// TwinCAT 3 PLC project Plc_Prog
// ProgramVersion: 3.1.4024.0
// libraries:
//   CPNTeck - OSCAT BASIC, * (CPNTeck - Automação Industrial)
//   Tc2_EtherCAT, * (Beckhoff Automation GmbH)
//   Tc2_ModbusSrv, * (Beckhoff Automation GmbH)
//   Tc2_Standard, * (Beckhoff Automation GmbH)
//   Tc2_SUPS, * (Beckhoff Automation GmbH)
//   Tc2_System, * (Beckhoff Automation GmbH)
//   Tc2_Utilities, * (Beckhoff Automation GmbH)
//   Tc3_Module, * (Beckhoff Automation GmbH)
// project tree:
//   Function Blocks/DELTA - MS300/ C2000_ANALOG_INPUTS.TcDUT, C2000_ANALOG_OUTPUTS.TcDUT, C2000_CONTROLWORD.TcDUT, C2000_DEV_CONFIG.TcDUT (not stored), C2000_DIGITAL_INPUTS.TcDUT (not stored), C2000_DIGITAL_OUTPUTS.TcDUT, C2000_DRVTOPLC_PDOS.TcDUT, C2000_PDOS.TcDUT (not stored), C2000_PLCTODRV_PDOS.TcDUT, C2000_STATUSWORD.TcDUT, E_C2000_ModeOfOperation.TcDUT (not stored), FB_DELTA_C2000_ETC.TcPOU
//   Function Blocks/IOs/Beckhoff/Common/ FB_SavePersistentData.TcPOU
//   Function Blocks/IOs/Beckhoff/EL1809 - Digital Inputs/DataTypes/ EL1809_DEV_CONFIG.TcDUT (not stored), EL1809_HWTOPLC_PDOS.TcDUT, EL1809_PDOS.TcDUT (not stored)
//   Function Blocks/IOs/Beckhoff/EL1809 - Digital Inputs/ FB_EL1809.TcPOU (not stored)
//   Function Blocks/IOs/Beckhoff/EL3052 - Ai 2 x 4-20MA - 12bit/DataTypes/ EL3052_DEV_CONFIG.TcDUT, EL3052_DEV_STATUS.TcDUT, EL3052_HWTOPLC_PDOS.TcDUT, EL3052_CHANNEL.TcDUT (not stored), EL3052_PDOS.TcDUT (not stored)
//   Function Blocks/IOs/Beckhoff/EL3052 - Ai 2 x 4-20MA - 12bit/ FB_EL3052.TcPOU
//   Function Blocks/IOs/Beckhoff/EL2809 - Digital Outputs/DataTypes/ EL2809_DEV_CONFIG.TcDUT, EL2809_PDOS.TcDUT (not stored), EL2809_PLCTOHW_PDOS.TcDUT
//   Function Blocks/IOs/Beckhoff/EL2809 - Digital Outputs/ FB_EL2809.TcPOU (not stored)
//   Function Blocks/IOs/Beckhoff/EL3152 - Ai 2 x 4-20MA - 16bit/DataTypes/ EL3152_CHANNEL.TcDUT, EL3152_DEV_CONFIG.TcDUT, EL3152_DEV_STATUS.TcDUT, EL3152_HWTOPLC_PDOS.TcDUT (not stored), EL3152_PDOS.TcDUT
//   Function Blocks/IOs/Beckhoff/EL3152 - Ai 2 x 4-20MA - 16bit/ FB_EL3152.TcPOU (not stored)
//   Function Blocks/IOs/Beckhoff/EL3154 - Ai 4 x 4-20MA - 16bit/DataTypes/ EL3154_CHANNEL.TcDUT (not stored), EL3154_DEV_CONFIG.TcDUT, EL3154_DEV_STATUS.TcDUT, EL3154_HWTOPLC_PDOS.TcDUT (not stored), EL3154_PDOS.TcDUT
//   Function Blocks/IOs/Beckhoff/EL3154 - Ai 4 x 4-20MA - 16bit/ FB_EL3154.TcPOU
//   Function Blocks/IOs/Beckhoff/EL3204 - Ai 4 x PT100 %28RTD%29/DataTypes/ EL3204_DEV_CONFIG.TcDUT (not stored), EL3204_CHANNEL.TcDUT (not stored), EL3204_DEV_STATUS.TcDUT (not stored), EL3204_HWTOPLC_PDOS.TcDUT (not stored), EL3204_PDOS.TcDUT (not stored)
//   Function Blocks/IOs/Beckhoff/EL3204 - Ai 4 x PT100 %28RTD%29/ FB_EL3204.TcPOU (not stored)
//   Function Blocks/IOs/Beckhoff/EL4004 - AQ 4 x 0-10V/DataTypes/ EL4004_DEV_CONFIG.TcDUT, EL4004_HWTOPLC_PDOS.TcDUT, EL4004_PDOS.TcDUT
//   Function Blocks/IOs/Beckhoff/EL4004 - AQ 4 x 0-10V/ FB_EL4004.TcPOU
//   Function Blocks/IOs/Beckhoff/EL4024 - AQ 4 x 4-20MA/DataTypes/ EL4024_DEV_CONFIG.TcDUT, EL4024_HWTOPLC_PDOS.TcDUT, EL4024_PDOS.TcDUT
//   Function Blocks/IOs/Beckhoff/EL4024 - AQ 4 x 4-20MA/ FB_EL4024.TcPOU
//   Function Blocks/IOs/Beckhoff/EL6910 - TwinSAFE PLC/ EL6910_ESTOP.TcDUT, EL6910_ESTOP_DIGNOSTICS.TcDUT, EL6910_ESTOP_STATUS.TcDUT (not stored), EL6910_HWTOPLC_PDOS.TcDUT, EL6910_PDOS.TcDUT (not stored), EL6910_PLCTOHW_PDOS.TcDUT (not stored), FB_EL6910.TcPOU
//   Function Blocks/PaperMachine/Auxiliary/ FB_FormingBoardDriveControl.TcPOU (not stored), FB_ConsistencyControllerModbusTcp.TcPOU, FB_FormingBoardRollUpDown.TcPOU (not stored), FB_FormingBoardWireStretchControl.TcPOU, FB_Gen_SRamp.TcPOU, FB_HeadboxLipsPWMControl.TcPOU, FB_JumboWeightCapture.TcPOU, FB_LevelControl.TcPOU (not stored), FB_LevelControl_V2.TcPOU, FB_MixPumpControl.TcPOU (not stored), FB_MixPumpControl_V1.TcPOU (not stored), FB_PaperMachine.TcPOU (not stored), FB_PressureControl.TcPOU, FB_PressureControl_V1.TcPOU (not stored), FB_StockPumpFlowControl.TcPOU, FB_VfdProcessControler.TcPOU (not stored), FB_ValveProcessControler.TcPOU, FB_SimpleMotorStart.TcPOU (not stored), FB_SimpleMotorStart_V2.TcPOU (not stored), FB_SimpleMotorStart_V3.TcPOU, FB_SoftstarterSimple.TcPOU, FB_SoftstarterWithBypass.TcPOU (not stored), FB_SoftstarterWithBypass_V1.TcPOU (not stored), FB_SpeedDroopControl.TcPOU (not stored), FB_SpeedDroopControl_1.TcPOU (not stored), FB_WirePitControl.TcPOU, FB_WirePitControl_1.TcPOU
//   Function Blocks/PaperMachine/DataTypes/ PaperMachine_TypeHmiConfig.TcDUT, PaperMachine_TypeHmiCommands.TcDUT, PaperMachine_TypeHmiStatus.TcDUT, PaperMachine_TypeHmiAlarms.TcDUT, ST_ConsistencyControllerConfig.TcDUT, ST_ConsistencyControllerInputs.TcDUT
//   Function Blocks/PaperMachine/DriveControl/ FB_DryingSectionDriveControl_V1.TcPOU, FB_DryingSectionDriveControl_V2.TcPOU, FB_DryingSectionDriveControl_V3.TcPOU (not stored), FB_FormingBoardControl_V3.TcPOU, FB_PressSectionDriveControl_V2_bak.TcPOU (not stored), FB_WinderDriveControl_V1.TcPOU (not stored), FB_DryingSectionLubrificationControl_V1.TcPOU (not stored), FB_DryingSectionPressureControl.TcPOU, FB_FormingBoardControl_V1.TcPOU (not stored), FB_PressSectionDriveControl_V1.TcPOU, FB_PressSectionDriveControl_V2.TcPOU
//   Function Blocks/PaperMachine/ FB_AlarmControl.TcPOU (not stored), FB_GroupDisplayFilters_V1.TcPOU (not stored), FB_GroupDriveControl_V1.TcPOU, FB_GroupSpeedControl_V1.TcPOU (not stored), FB_FormingBoardSpeedControl.TcPOU, FB_DryingSecSpeedControl.TcPOU (not stored), FB_WinderSpeedControl.TcPOU (not stored), FB_GroupTorqueTrimControl_V1.TcPOU (not stored), FB_GroupTorqueTrimControl_V2.TcPOU
//   Function Blocks/Rewinder/DataTypes/ RewinderConfig_TypeStruct.TcDUT, Rewinder_TypePressRoll.TcDUT (not stored), Rewinder_TypeBrakeControl.TcDUT (not stored)
//   Function Blocks/Rewinder/ FB_RewinderControl_V1.TcPOU
//   GVLs/ GVL_Hw.TcGVL
//   / PlcTask.TcTTO, RecipeManager.TcRMO (not stored)
//   POUs/Implicit Checks/ CheckBounds.TcPOU, CheckDivDInt.TcPOU (not stored), CheckDivLInt.TcPOU (not stored), CheckDivLReal.TcPOU, CheckDivReal.TcPOU, CheckLRangeSigned.TcPOU, CheckLRangeUnsigned.TcPOU, CheckPointer.TcPOU, CheckRangeSigned.TcPOU, CheckRangeUnsigned.TcPOU (not stored)
//   POUs/ MAIN.TcPOU
// real-time tasks:
//   TASK PlcTask: cycle T#5ms, priority 20, ADS port 350
// I/O:
//   DEVICE ETH, AmsNetId 192.168.100.1.3.1
//     +P5=050-BC1 - PLC Cabinet [EK1100 EtherCAT Coupler (2A E-Bus)]
//       +P5=050-DI1 (EL1809) [EL1809 16Ch. Dig. Input 24V, 3ms]
//       +P5=050-DI2 (EL1809) [EL1809 16Ch. Dig. Input 24V, 3ms]
//       +P5=050-DI3 (EL1809) [EL1809 16Ch. Dig. Input 24V, 3ms]
//       +P5=050-DO1 (EL2809) [EL2809 16Ch. Dig. Output 24V, 0.5A]
//       +P5=050-DO2 (EL2809) [EL2809 16Ch. Dig. Output 24V, 0.5A]
//       +P5=050-DO3 (EL2809) [EL2809 16Ch. Dig. Output 24V, 0.5A]
//       +P5=050-SP1 (EL6910) [EL6910, TwinSAFE PLC]
//       +P5=050-SI1 (EL1918) [EL1918, 8Ch. Safety Input 24V, TwinSAFE]
//         modules: Module 1 (FSOE), Module 2 (FSLOGIC)
//       +P5=050-SO1 (EL2904) [EL2904, 4 Ch. Safety Output 24V, 0.5A, TwinSAFE]
//         modules: Module 1 (FSOES), Module 2 (DO)
//       +P5=050-SO2 (EL2904) [EL2904, 4 Ch. Safety Output 24V, 0.5A, TwinSAFE]
//         modules: Module 1 (FSOES), Module 2 (DO)
//       +P5=050-BC2 [EL6601 1 Port Switch (Ethernet, CoE)]
//       +P5=050-BC3 [EL6601 1 Port Switch (Ethernet, CoE)]
//       +P5=050-BE1 [EL9011 End Terminal]
//     +P5=050-BC2 - PLC Cabinet [EK1100 EtherCAT Coupler (2A E-Bus)]
//       +P5=050-AI (EL3052) [EL3052 2Ch. Ana. Input 4-20mA]
//       +P5=050-AI2 (EL3152) [EL3152 2Ch. Ana Input 4-20mA]
//       +P5=050-AI3 (EL3052) [EL3052 2Ch. Ana. Input 4-20mA]
//       +P5=050-AI4 (EL3052) [EL3052 2Ch. Ana. Input 4-20mA]
//       +P5=050-BE2 [EL9011 End Terminal]
//     +P4=300-UG1 - Mix Pump [Delta CH2000 EtherCAT(CoE)]
//     +P3=300-UG1 - WirePit Pump [Delta CH2000 EtherCAT(CoE)]
//     +P3=100-UG1 - SuctionRoll [Delta CH2000 EtherCAT(CoE)]
//     +P3=100-UG1 - CouchPit [Delta CH2000 EtherCAT(CoE)]
//     +P3=100-UG2 - Stock pump [Delta CH2000 EtherCAT(CoE)]
//     +P2=100-UG1 - Drive Roll [Delta CH2000 EtherCAT(CoE)]
//     +P9=050-BC1 - Vaccum PLC Cabinet [EK1100 EtherCAT Coupler (2A E-Bus)]
//       +P9=050-DI1 (EL1809) [EL1809 16Ch. Dig. Input 24V, 3ms]
//       +P9=050-DI2 (EL1809) [EL1809 16Ch. Dig. Input 24V, 3ms]
//       +P9=050-DI3 (EL1809) [EL1809 16Ch. Dig. Input 24V, 3ms]
//       +P9=050-DO1 (EL2809) [EL2809 16Ch. Dig. Output 24V, 0.5A]
//       +P9=050-DO2 (EL2809) [EL2809 16Ch. Dig. Output 24V, 0.5A]
//       +P9=050-DO3 (EL2809) [EL2809 16Ch. Dig. Output 24V, 0.5A]
//       +P9=050-AI1 (EL3054) [EL3054 4Ch. Ana. Input 4-20mA]
//       Term 101 (EL3052) [EL3052 2Ch. Ana. Input 4-20mA]
//       Term 102 (EL4004) [EL4004 4Ch. Ana. Output 0-10V, 12bit]
//       Term 151 (EL9011) [EL9011 End Terminal]
//       +P9=050-BE1 [EL9011 End Terminal]
//     +P10=050-BC1 - Press / Dryer PLC Cabinet [EK1100 EtherCAT Coupler (2A E-Bus)]
//       +P10=050-DI1 (EL1809) [EL1809 16Ch. Dig. Input 24V, 3ms]
//       +P10=050-DI2 (EL1809) [EL1809 16Ch. Dig. Input 24V, 3ms]
//       +P10=050-DI3 (EL1809) [EL1809 16Ch. Dig. Input 24V, 3ms]
//       +P10=050-DI4 (EL1809) [EL1809 16Ch. Dig. Input 24V, 3ms]
//       +P10=050-DI5 (EL1809) [EL1809 16Ch. Dig. Input 24V, 3ms]
//       +P10=050-DI6 (EL1809) [EL1809 16Ch. Dig. Input 24V, 3ms]
//       +P10=050-DI7 (EL1809) [EL1809 16Ch. Dig. Input 24V, 3ms]
//       +P10=050-DI8 (EL1809) [EL1809 16Ch. Dig. Input 24V, 3ms]
//       +P10=050-DO1 (EL2809) [EL2809 16Ch. Dig. Output 24V, 0.5A]
//       +P10=050-DO2 (EL2809) [EL2809 16Ch. Dig. Output 24V, 0.5A]
//       +P10=050-DO3 (EL2809) [EL2809 16Ch. Dig. Output 24V, 0.5A]
//       +P10=050-DO4 (EL2809) [EL2809 16Ch. Dig. Output 24V, 0.5A]
//       +P10=050-SI1 (EL1918) [EL1918, 8Ch. Safety Input 24V, TwinSAFE]
//         modules: Module 1 (FSOE), Module 2 (FSLOGIC)
//       +P10=050-SO1 (EL2904) [EL2904, 4 Ch. Safety Output 24V, 0.5A, TwinSAFE]
//         modules: Module 1 (FSOES), Module 2 (DO)
//       +P10=050-BE1 [EL9011 End Terminal]
//     +P10=050-BC2 - Press / Dryer PLC Cabinet [EK1100 EtherCAT Coupler (2A E-Bus)]
//       +P10=050-AI1 (EL3054) [EL3054 4Ch. Ana. Input 4-20mA]
//       +P10=050-AI2 (EL3204) [EL3204 4Ch. Ana. Input PT100 (RTD)]
//       +P10=050-AO1(EL4024) [EL4024 4Ch. Ana. Output 4-20mA, 12bit]
//       +P10=050-BE2 [EL9011 End Terminal]
//     +P11=400-UG1 - Second Press [Delta C2000Plus EtherCAT(CoE)]
//     +P12=400-UG1 - First Press [Delta C2000Plus EtherCAT(CoE)]
//     +P13=500-UG1 - Dryer Section GR1 - Upper GR1 Slave [Delta C2000Plus EtherCAT(CoE)]
//     +P12=500-UG2 - Dryer Section GR1 - Lower GR1 Master [Delta C2000Plus EtherCAT(CoE)]
//     +P12=500-UG3 - Dryer Section GR1 - Upper Master [Delta CH2000 EtherCAT(CoE)]
//     +P12=501-UG1 - Dryer Section  GR2 - Lower Slave [Delta C2000Plus EtherCAT(CoE)]
//     +P12=501-UG2 - Dryer Section GR2 - Upper Slave [Delta CH2000 EtherCAT(CoE)]
//     +P12=501-UG3 - Dryer Section GR2 - Lower Master [Delta C2000Plus EtherCAT(CoE)]
//     +P13=501-UG1 - Dryer Section GR2 - Upper Master [Delta CH2000 EtherCAT(CoE)]
//     +P13=502-UG2 - Dryer Section GR3 - Lower Slave [Delta C2000Plus EtherCAT(CoE)]
//     +P13=502-UG2 - Dryer Section GR3 - Upper Slave [Delta C2000Plus EtherCAT(CoE)]
//     +P13=502-UG3 - Dryer Section GR3 - Lower Master [Delta C2000Plus EtherCAT(CoE)]
//     +P13=502-UG4 - Dryer Section GR3 - Upper Master [Delta C2000Plus EtherCAT(CoE)]
//     +P14=600-UG1 - Winder [Delta C2000Plus EtherCAT(CoE)]
//     +CP2=050-BC1 - Winder command panel [EK1100 EtherCAT Coupler (2A E-Bus)]
//       +CP2=050-SI1 (EL1918) [EL1918, 8Ch. Safety Input 24V, TwinSAFE]
//         modules: Module 1 (FSOE), Module 2 (FSLOGIC)
//       +CP2=050-DI1 (EL1809) [EL1809 16Ch. Dig. Input 24V, 3ms]
//       +CP2=050-DO1 (EL2809 [EL2809 16Ch. Dig. Output 24V, 0.5A]
//       +CP2=050-AO1 (EL4024) [EL4024 4Ch. Ana. Output 4-20mA, 12bit]
//       +CP2=050-BE1 (EL4024) [EL9011 End Terminal]
// variable links:
//   ETH <-> ETH/+CP2=050-BC1 - Winder command panel/+CP2=050-SI1 (EL1918)
//     +P5=050-BC1 - PLC Cabinet/+P5=050-SP1 (EL6910)/ConnectionInputs/TwinSafeGroup1.+CP2=050-SI1 (EL1918) - Module 1 (FSOE)_9 TxPDO <-> Module 1 (FSOE)/FSoE Outputs/FSOE
//     +P5=050-BC1 - PLC Cabinet/+P5=050-SP1 (EL6910)/ConnectionOutputs/TwinSafeGroup1.+CP2=050-SI1 (EL1918) - Module 1 (FSOE)_9 RxPDO <-> Module 1 (FSOE)/FSoE Inputs/FSOE
//   ETH <-> ETH/+P10=050-BC1 - Press / Dryer PLC Cabinet/+P10=050-SI1 (EL1918)
//     +P5=050-BC1 - PLC Cabinet/+P5=050-SP1 (EL6910)/ConnectionInputs/TwinSafeGroup1.+P10=050-SI1 (EL1918) - Module 1 (FSOE)_7 TxPDO <-> Module 1 (FSOE)/FSoE Outputs/FSOE
//   ETH <-> ETH/+P10=050-BC1 - Press / Dryer PLC Cabinet/+P10=050-SO1 (EL2904)
//     +P5=050-BC1 - PLC Cabinet/+P5=050-SP1 (EL6910)/ConnectionInputs/TwinSafeGroup1.+P10=050-SO1 (EL2904) - Module 1 (FSOES)_8 TxPDO <-> Module 1 (FSOES)/RxPDO/FSOE
//     +P5=050-BC1 - PLC Cabinet/+P5=050-SP1 (EL6910)/ConnectionOutputs/TwinSafeGroup1.+P10=050-SO1 (EL2904) - Module 1 (FSOES)_8 RxPDO <-> Module 1 (FSOES)/TxPDO/FSOE
//   ETH <-> ETH/+P5=050-BC1 - PLC Cabinet/+P5=050-SI1 (EL1918)
//     +P5=050-BC1 - PLC Cabinet/+P5=050-SP1 (EL6910)/ConnectionInputs/TwinSafeGroup1.Term 9 (EL1918) - Module 1 (FSOE)_3 TxPDO <-> Module 1 (FSOE)/FSoE Outputs/FSOE
//   ETH <-> ETH/+P5=050-BC1 - PLC Cabinet/+P5=050-SP1 (EL6910)
//     +P10=050-BC1 - Press / Dryer PLC Cabinet/+P10=050-SI1 (EL1918)/Module 1 (FSOE)/FSoE Inputs/FSOE <-> ConnectionOutputs/TwinSafeGroup1.+P10=050-SI1 (EL1918) - Module 1 (FSOE)_7 RxPDO
//     +P5=050-BC1 - PLC Cabinet/+P5=050-SI1 (EL1918)/Module 1 (FSOE)/FSoE Inputs/FSOE <-> ConnectionOutputs/TwinSafeGroup1.Term 9 (EL1918) - Module 1 (FSOE)_3 RxPDO
//     +P5=050-BC1 - PLC Cabinet/+P5=050-SO1 (EL2904)/Module 1 (FSOES)/RxPDO/FSOE <-> ConnectionInputs/TwinSafeGroup1.Term 10 (EL2904) - Module 1 (FSOES)_4 TxPDO
//     +P5=050-BC1 - PLC Cabinet/+P5=050-SO2 (EL2904)/Module 1 (FSOES)/RxPDO/FSOE <-> ConnectionInputs/TwinSafeGroup1.Term 11 (EL2904) - Module 1 (FSOES)_5 TxPDO
//     +P5=050-BC1 - PLC Cabinet/+P5=050-SO1 (EL2904)/Module 1 (FSOES)/TxPDO/FSOE <-> ConnectionOutputs/TwinSafeGroup1.Term 10 (EL2904) - Module 1 (FSOES)_4 RxPDO
//     +P5=050-BC1 - PLC Cabinet/+P5=050-SO2 (EL2904)/Module 1 (FSOES)/TxPDO/FSOE <-> ConnectionOutputs/TwinSafeGroup1.Term 11 (EL2904) - Module 1 (FSOES)_5 RxPDO
//   Plc_Prog/Plc_Prog Instance <-> ETH/+CP2=050-BC1 - Winder command panel/+CP2=050-AO1 (EL4024)
//     PlcTask Outputs/.CP1_050_AO1.PDOS.HwToPLC.Channel1 <-> AO Outputs Channel 1/Analog output
//     PlcTask Outputs/.CP1_050_AO1.PDOS.HwToPLC.Channel2 <-> AO Outputs Channel 2/Analog output
//     PlcTask Outputs/.CP1_050_AO1.PDOS.HwToPLC.Channel3 <-> AO Outputs Channel 3/Analog output
//     PlcTask Outputs/.CP1_050_AO1.PDOS.HwToPLC.Channel4 <-> AO Outputs Channel 4/Analog output
//   Plc_Prog/Plc_Prog Instance <-> ETH/+CP2=050-BC1 - Winder command panel/+CP2=050-DI1 (EL1809)
//     PlcTask Inputs/.CP1_050_DI1.PDOS.digitalInput_01 <-> Channel 1/Input
//     PlcTask Inputs/.CP1_050_DI1.PDOS.digitalInput_02 <-> Channel 2/Input
//     PlcTask Inputs/.CP1_050_DI1.PDOS.digitalInput_03 <-> Channel 3/Input
//     PlcTask Inputs/.CP1_050_DI1.PDOS.digitalInput_04 <-> Channel 4/Input
//     PlcTask Inputs/.CP1_050_DI1.PDOS.digitalInput_05 <-> Channel 5/Input
//     PlcTask Inputs/.CP1_050_DI1.PDOS.digitalInput_06 <-> Channel 6/Input
//     PlcTask Inputs/.CP1_050_DI1.PDOS.digitalInput_07 <-> Channel 7/Input
//     PlcTask Inputs/.CP1_050_DI1.PDOS.digitalInput_08 <-> Channel 8/Input
//     PlcTask Inputs/.CP1_050_DI1.PDOS.digitalInput_09 <-> Channel 9/Input
//     PlcTask Inputs/.CP1_050_DI1.PDOS.digitalInput_10 <-> Channel 10/Input
//     PlcTask Inputs/.CP1_050_DI1.PDOS.digitalInput_11 <-> Channel 11/Input
//     PlcTask Inputs/.CP1_050_DI1.PDOS.digitalInput_12 <-> Channel 12/Input
//     PlcTask Inputs/.CP1_050_DI1.PDOS.digitalInput_13 <-> Channel 13/Input
//     PlcTask Inputs/.CP1_050_DI1.PDOS.digitalInput_14 <-> Channel 14/Input
//     PlcTask Inputs/.CP1_050_DI1.PDOS.digitalInput_15 <-> Channel 15/Input
//     PlcTask Inputs/.CP1_050_DI1.PDOS.digitalInput_16 <-> Channel 16/Input
//   Plc_Prog/Plc_Prog Instance <-> ETH/+CP2=050-BC1 - Winder command panel/+CP2=050-DO1 (EL2809
//     PlcTask Outputs/.CP1_050_DO1.PDOS.PlcToHw.digitalOutput_01 <-> Channel 1/Output
//     PlcTask Outputs/.CP1_050_DO1.PDOS.PlcToHw.digitalOutput_02 <-> Channel 2/Output
//     PlcTask Outputs/.CP1_050_DO1.PDOS.PlcToHw.digitalOutput_03 <-> Channel 3/Output
//     PlcTask Outputs/.CP1_050_DO1.PDOS.PlcToHw.digitalOutput_04 <-> Channel 4/Output
//     PlcTask Outputs/.CP1_050_DO1.PDOS.PlcToHw.digitalOutput_05 <-> Channel 5/Output
//     PlcTask Outputs/.CP1_050_DO1.PDOS.PlcToHw.digitalOutput_06 <-> Channel 6/Output
//     PlcTask Outputs/.CP1_050_DO1.PDOS.PlcToHw.digitalOutput_07 <-> Channel 7/Output
//     PlcTask Outputs/.CP1_050_DO1.PDOS.PlcToHw.digitalOutput_08 <-> Channel 8/Output
//     PlcTask Outputs/.CP1_050_DO1.PDOS.PlcToHw.digitalOutput_09 <-> Channel 9/Output
//     PlcTask Outputs/.CP1_050_DO1.PDOS.PlcToHw.digitalOutput_10 <-> Channel 10/Output
//     PlcTask Outputs/.CP1_050_DO1.PDOS.PlcToHw.digitalOutput_11 <-> Channel 11/Output
//     PlcTask Outputs/.CP1_050_DO1.PDOS.PlcToHw.digitalOutput_12 <-> Channel 12/Output
//     PlcTask Outputs/.CP1_050_DO1.PDOS.PlcToHw.digitalOutput_13 <-> Channel 13/Output
//     PlcTask Outputs/.CP1_050_DO1.PDOS.PlcToHw.digitalOutput_14 <-> Channel 14/Output
//     PlcTask Outputs/.CP1_050_DO1.PDOS.PlcToHw.digitalOutput_15 <-> Channel 15/Output
//     PlcTask Outputs/.CP1_050_DO1.PDOS.PlcToHw.digitalOutput_16 <-> Channel 16/Output
//   Plc_Prog/Plc_Prog Instance <-> ETH/+P10=050-BC1 - Press / Dryer PLC Cabinet/+P10=050-DI1 (EL1809)
//     PlcTask Inputs/.P10_050_DI1.PDOS.digitalInput_01 <-> Channel 1/Input
//     PlcTask Inputs/.P10_050_DI1.PDOS.digitalInput_02 <-> Channel 2/Input
//     PlcTask Inputs/.P10_050_DI1.PDOS.digitalInput_03 <-> Channel 3/Input
//     PlcTask Inputs/.P10_050_DI1.PDOS.digitalInput_04 <-> Channel 4/Input
//     PlcTask Inputs/.P10_050_DI1.PDOS.digitalInput_05 <-> Channel 5/Input
//     PlcTask Inputs/.P10_050_DI1.PDOS.digitalInput_06 <-> Channel 6/Input
//     PlcTask Inputs/.P10_050_DI1.PDOS.digitalInput_07 <-> Channel 7/Input
//     PlcTask Inputs/.P10_050_DI1.PDOS.digitalInput_08 <-> Channel 8/Input
//     PlcTask Inputs/.P10_050_DI1.PDOS.digitalInput_09 <-> Channel 9/Input
//     PlcTask Inputs/.P10_050_DI1.PDOS.digitalInput_10 <-> Channel 10/Input
//     PlcTask Inputs/.P10_050_DI1.PDOS.digitalInput_11 <-> Channel 11/Input
//     PlcTask Inputs/.P10_050_DI1.PDOS.digitalInput_12 <-> Channel 12/Input
//     PlcTask Inputs/.P10_050_DI1.PDOS.digitalInput_13 <-> Channel 13/Input
//     PlcTask Inputs/.P10_050_DI1.PDOS.digitalInput_14 <-> Channel 14/Input
//     PlcTask Inputs/.P10_050_DI1.PDOS.digitalInput_15 <-> Channel 15/Input
//     PlcTask Inputs/.P10_050_DI1.PDOS.digitalInput_16 <-> Channel 16/Input
//   Plc_Prog/Plc_Prog Instance <-> ETH/+P10=050-BC1 - Press / Dryer PLC Cabinet/+P10=050-DI2 (EL1809)
//     PlcTask Inputs/.P10_050_DI2.PDOS.digitalInput_01 <-> Channel 1/Input
//     PlcTask Inputs/.P10_050_DI2.PDOS.digitalInput_02 <-> Channel 2/Input
//     PlcTask Inputs/.P10_050_DI2.PDOS.digitalInput_03 <-> Channel 3/Input
//     PlcTask Inputs/.P10_050_DI2.PDOS.digitalInput_04 <-> Channel 4/Input
//     PlcTask Inputs/.P10_050_DI2.PDOS.digitalInput_05 <-> Channel 5/Input
//     PlcTask Inputs/.P10_050_DI2.PDOS.digitalInput_06 <-> Channel 6/Input
//     PlcTask Inputs/.P10_050_DI2.PDOS.digitalInput_07 <-> Channel 7/Input
//     PlcTask Inputs/.P10_050_DI2.PDOS.digitalInput_08 <-> Channel 8/Input
//     PlcTask Inputs/.P10_050_DI2.PDOS.digitalInput_09 <-> Channel 9/Input
//     PlcTask Inputs/.P10_050_DI2.PDOS.digitalInput_10 <-> Channel 10/Input
//     PlcTask Inputs/.P10_050_DI2.PDOS.digitalInput_12 <-> Channel 12/Input
//     PlcTask Inputs/.P10_050_DI2.PDOS.digitalInput_13 <-> Channel 13/Input
//     PlcTask Inputs/.P10_050_DI2.PDOS.digitalInput_14 <-> Channel 14/Input
//     PlcTask Inputs/.P10_050_DI2.PDOS.digitalInput_15 <-> Channel 15/Input
//     PlcTask Inputs/.P10_050_DI2.PDOS.digitalInput_16 <-> Channel 16/Input
//     PlcTask Inputs/.P10_050_DI2.PDOS.digitalInput_11 <-> Channel 11/.P10_050_DI2.PDOS.digitalInput_11
//   Plc_Prog/Plc_Prog Instance <-> ETH/+P10=050-BC1 - Press / Dryer PLC Cabinet/+P10=050-DI3 (EL1809)
//     PlcTask Inputs/.P10_050_DI3.PDOS.digitalInput_01 <-> Channel 1/Input
//     PlcTask Inputs/.P10_050_DI3.PDOS.digitalInput_02 <-> Channel 2/Input
//     PlcTask Inputs/.P10_050_DI3.PDOS.digitalInput_03 <-> Channel 3/Input
//     PlcTask Inputs/.P10_050_DI3.PDOS.digitalInput_04 <-> Channel 4/Input
//     PlcTask Inputs/.P10_050_DI3.PDOS.digitalInput_05 <-> Channel 5/Input
//     PlcTask Inputs/.P10_050_DI3.PDOS.digitalInput_06 <-> Channel 6/Input
//     PlcTask Inputs/.P10_050_DI3.PDOS.digitalInput_07 <-> Channel 7/Input
//     PlcTask Inputs/.P10_050_DI3.PDOS.digitalInput_08 <-> Channel 8/Input
//     PlcTask Inputs/.P10_050_DI3.PDOS.digitalInput_09 <-> Channel 9/Input
//     PlcTask Inputs/.P10_050_DI3.PDOS.digitalInput_10 <-> Channel 10/Input
//     PlcTask Inputs/.P10_050_DI3.PDOS.digitalInput_11 <-> Channel 11/Input
//     PlcTask Inputs/.P10_050_DI3.PDOS.digitalInput_12 <-> Channel 12/Input
//     PlcTask Inputs/.P10_050_DI3.PDOS.digitalInput_13 <-> Channel 13/Input
//     PlcTask Inputs/.P10_050_DI3.PDOS.digitalInput_14 <-> Channel 14/Input
//     PlcTask Inputs/.P10_050_DI3.PDOS.digitalInput_15 <-> Channel 15/Input
//     PlcTask Inputs/.P10_050_DI3.PDOS.digitalInput_16 <-> Channel 16/Input
//   Plc_Prog/Plc_Prog Instance <-> ETH/+P10=050-BC1 - Press / Dryer PLC Cabinet/+P10=050-DI4 (EL1809)
//     PlcTask Inputs/.P10_050_DI4.PDOS.digitalInput_01 <-> Channel 1/Input
//     PlcTask Inputs/.P10_050_DI4.PDOS.digitalInput_02 <-> Channel 2/Input
//     PlcTask Inputs/.P10_050_DI4.PDOS.digitalInput_03 <-> Channel 3/Input
//     PlcTask Inputs/.P10_050_DI4.PDOS.digitalInput_04 <-> Channel 4/Input
//     PlcTask Inputs/.P10_050_DI4.PDOS.digitalInput_05 <-> Channel 5/Input
//     PlcTask Inputs/.P10_050_DI4.PDOS.digitalInput_06 <-> Channel 6/Input
//     PlcTask Inputs/.P10_050_DI4.PDOS.digitalInput_07 <-> Channel 7/Input
//     PlcTask Inputs/.P10_050_DI4.PDOS.digitalInput_08 <-> Channel 8/Input
//     PlcTask Inputs/.P10_050_DI4.PDOS.digitalInput_09 <-> Channel 9/Input
//     PlcTask Inputs/.P10_050_DI4.PDOS.digitalInput_10 <-> Channel 10/Input
//     PlcTask Inputs/.P10_050_DI4.PDOS.digitalInput_11 <-> Channel 11/Input
//     PlcTask Inputs/.P10_050_DI4.PDOS.digitalInput_12 <-> Channel 12/Input
//     PlcTask Inputs/.P10_050_DI4.PDOS.digitalInput_13 <-> Channel 13/Input
//     PlcTask Inputs/.P10_050_DI4.PDOS.digitalInput_14 <-> Channel 14/Input
//     PlcTask Inputs/.P10_050_DI4.PDOS.digitalInput_15 <-> Channel 15/Input
//     PlcTask Inputs/.P10_050_DI4.PDOS.digitalInput_16 <-> Channel 16/Input
//   Plc_Prog/Plc_Prog Instance <-> ETH/+P10=050-BC1 - Press / Dryer PLC Cabinet/+P10=050-DI5 (EL1809)
//     PlcTask Inputs/.P10_050_DI5.PDOS.digitalInput_01 <-> Channel 1/Input
//     PlcTask Inputs/.P10_050_DI5.PDOS.digitalInput_02 <-> Channel 2/Input
//     PlcTask Inputs/.P10_050_DI5.PDOS.digitalInput_03 <-> Channel 3/Input
//     PlcTask Inputs/.P10_050_DI5.PDOS.digitalInput_04 <-> Channel 4/Input
//     PlcTask Inputs/.P10_050_DI5.PDOS.digitalInput_05 <-> Channel 5/Input
//     PlcTask Inputs/.P10_050_DI5.PDOS.digitalInput_06 <-> Channel 6/Input
//     PlcTask Inputs/.P10_050_DI5.PDOS.digitalInput_07 <-> Channel 7/Input
//     PlcTask Inputs/.P10_050_DI5.PDOS.digitalInput_08 <-> Channel 8/Input
//     PlcTask Inputs/.P10_050_DI5.PDOS.digitalInput_09 <-> Channel 9/Input
//     PlcTask Inputs/.P10_050_DI5.PDOS.digitalInput_10 <-> Channel 10/Input
//     PlcTask Inputs/.P10_050_DI5.PDOS.digitalInput_11 <-> Channel 11/Input
//     PlcTask Inputs/.P10_050_DI5.PDOS.digitalInput_12 <-> Channel 12/Input
//     PlcTask Inputs/.P10_050_DI5.PDOS.digitalInput_13 <-> Channel 13/Input
//     PlcTask Inputs/.P10_050_DI5.PDOS.digitalInput_14 <-> Channel 14/Input
//     PlcTask Inputs/.P10_050_DI5.PDOS.digitalInput_15 <-> Channel 15/Input
//     PlcTask Inputs/.P10_050_DI5.PDOS.digitalInput_16 <-> Channel 16/Input
//   Plc_Prog/Plc_Prog Instance <-> ETH/+P10=050-BC1 - Press / Dryer PLC Cabinet/+P10=050-DI6 (EL1809)
//     PlcTask Inputs/.P10_050_DI6.PDOS.digitalInput_01 <-> Channel 1/Input
//     PlcTask Inputs/.P10_050_DI6.PDOS.digitalInput_02 <-> Channel 2/Input
//     PlcTask Inputs/.P10_050_DI6.PDOS.digitalInput_03 <-> Channel 3/Input
//     PlcTask Inputs/.P10_050_DI6.PDOS.digitalInput_04 <-> Channel 4/Input
//     PlcTask Inputs/.P10_050_DI6.PDOS.digitalInput_05 <-> Channel 5/Input
//     PlcTask Inputs/.P10_050_DI6.PDOS.digitalInput_06 <-> Channel 6/Input
//     PlcTask Inputs/.P10_050_DI6.PDOS.digitalInput_07 <-> Channel 7/Input
//     PlcTask Inputs/.P10_050_DI6.PDOS.digitalInput_08 <-> Channel 8/Input
//     PlcTask Inputs/.P10_050_DI6.PDOS.digitalInput_09 <-> Channel 9/Input
//     PlcTask Inputs/.P10_050_DI6.PDOS.digitalInput_10 <-> Channel 10/Input
//     PlcTask Inputs/.P10_050_DI6.PDOS.digitalInput_11 <-> Channel 11/Input
//     PlcTask Inputs/.P10_050_DI6.PDOS.digitalInput_12 <-> Channel 12/Input
//     PlcTask Inputs/.P10_050_DI6.PDOS.digitalInput_13 <-> Channel 13/Input
//     PlcTask Inputs/.P10_050_DI6.PDOS.digitalInput_14 <-> Channel 14/Input
//     PlcTask Inputs/.P10_050_DI6.PDOS.digitalInput_15 <-> Channel 15/Input
//     PlcTask Inputs/.P10_050_DI6.PDOS.digitalInput_16 <-> Channel 16/Input
//   Plc_Prog/Plc_Prog Instance <-> ETH/+P10=050-BC1 - Press / Dryer PLC Cabinet/+P10=050-DI7 (EL1809)
//     PlcTask Inputs/.P10_050_DI7.PDOS.digitalInput_01 <-> Channel 1/Input
//     PlcTask Inputs/.P10_050_DI7.PDOS.digitalInput_02 <-> Channel 2/Input
//     PlcTask Inputs/.P10_050_DI7.PDOS.digitalInput_03 <-> Channel 3/Input
//     PlcTask Inputs/.P10_050_DI7.PDOS.digitalInput_04 <-> Channel 4/Input
//     PlcTask Inputs/.P10_050_DI7.PDOS.digitalInput_05 <-> Channel 5/Input
//     PlcTask Inputs/.P10_050_DI7.PDOS.digitalInput_06 <-> Channel 6/Input
//     PlcTask Inputs/.P10_050_DI7.PDOS.digitalInput_07 <-> Channel 7/Input
//     PlcTask Inputs/.P10_050_DI7.PDOS.digitalInput_08 <-> Channel 8/Input
//     PlcTask Inputs/.P10_050_DI7.PDOS.digitalInput_09 <-> Channel 9/Input
//     PlcTask Inputs/.P10_050_DI7.PDOS.digitalInput_10 <-> Channel 10/Input
//     PlcTask Inputs/.P10_050_DI7.PDOS.digitalInput_11 <-> Channel 11/Input
//     PlcTask Inputs/.P10_050_DI7.PDOS.digitalInput_12 <-> Channel 12/Input
//     PlcTask Inputs/.P10_050_DI7.PDOS.digitalInput_13 <-> Channel 13/Input
//     PlcTask Inputs/.P10_050_DI7.PDOS.digitalInput_14 <-> Channel 14/Input
//     PlcTask Inputs/.P10_050_DI7.PDOS.digitalInput_15 <-> Channel 15/Input
//     PlcTask Inputs/.P10_050_DI7.PDOS.digitalInput_16 <-> Channel 16/Input
//   Plc_Prog/Plc_Prog Instance <-> ETH/+P10=050-BC1 - Press / Dryer PLC Cabinet/+P10=050-DI8 (EL1809)
//     PlcTask Inputs/.P10_050_DI8.PDOS.digitalInput_01 <-> Channel 1/Input
//     PlcTask Inputs/.P10_050_DI8.PDOS.digitalInput_02 <-> Channel 2/Input
//     PlcTask Inputs/.P10_050_DI8.PDOS.digitalInput_03 <-> Channel 3/Input
//     PlcTask Inputs/.P10_050_DI8.PDOS.digitalInput_04 <-> Channel 4/Input
//     PlcTask Inputs/.P10_050_DI8.PDOS.digitalInput_05 <-> Channel 5/Input
//     PlcTask Inputs/.P10_050_DI8.PDOS.digitalInput_06 <-> Channel 6/Input
//     PlcTask Inputs/.P10_050_DI8.PDOS.digitalInput_07 <-> Channel 7/Input
//     PlcTask Inputs/.P10_050_DI8.PDOS.digitalInput_08 <-> Channel 8/Input
//     PlcTask Inputs/.P10_050_DI8.PDOS.digitalInput_09 <-> Channel 9/Input
//     PlcTask Inputs/.P10_050_DI8.PDOS.digitalInput_10 <-> Channel 10/Input
//     PlcTask Inputs/.P10_050_DI8.PDOS.digitalInput_11 <-> Channel 11/Input
//     PlcTask Inputs/.P10_050_DI8.PDOS.digitalInput_14 <-> Channel 14/Input
//     PlcTask Inputs/.P10_050_DI8.PDOS.digitalInput_16 <-> Channel 16/Input
//     PlcTask Inputs/.P10_050_DI8.PDOS.digitalInput_12 <-> Channel 12/Pressao Alta HPU
//     PlcTask Inputs/.P10_050_DI8.PDOS.digitalInput_13 <-> Channel 13/Pressao Baixa HPU
//     PlcTask Inputs/.P10_050_DI8.PDOS.digitalInput_15 <-> Channel 15/Nivel muito baixo HPU
//   Plc_Prog/Plc_Prog Instance <-> ETH/+P10=050-BC1 - Press / Dryer PLC Cabinet/+P10=050-DO1 (EL2809)
//     PlcTask Outputs/.P10_050_DO1.PDOS.PlcToHw.digitalOutput_01 <-> Channel 1/Output
//     PlcTask Outputs/.P10_050_DO1.PDOS.PlcToHw.digitalOutput_02 <-> Channel 2/Output
//     PlcTask Outputs/.P10_050_DO1.PDOS.PlcToHw.digitalOutput_03 <-> Channel 3/Output
//     PlcTask Outputs/.P10_050_DO1.PDOS.PlcToHw.digitalOutput_04 <-> Channel 4/Output
//     PlcTask Outputs/.P10_050_DO1.PDOS.PlcToHw.digitalOutput_05 <-> Channel 5/Output
//     PlcTask Outputs/.P10_050_DO1.PDOS.PlcToHw.digitalOutput_06 <-> Channel 6/Output
//     PlcTask Outputs/.P10_050_DO1.PDOS.PlcToHw.digitalOutput_07 <-> Channel 7/Output
//     PlcTask Outputs/.P10_050_DO1.PDOS.PlcToHw.digitalOutput_08 <-> Channel 8/Output
//     PlcTask Outputs/.P10_050_DO1.PDOS.PlcToHw.digitalOutput_09 <-> Channel 9/Output
//     PlcTask Outputs/.P10_050_DO1.PDOS.PlcToHw.digitalOutput_10 <-> Channel 10/Output
//     PlcTask Outputs/.P10_050_DO1.PDOS.PlcToHw.digitalOutput_11 <-> Channel 11/Output
//     PlcTask Outputs/.P10_050_DO1.PDOS.PlcToHw.digitalOutput_12 <-> Channel 12/Output
//     PlcTask Outputs/.P10_050_DO1.PDOS.PlcToHw.digitalOutput_13 <-> Channel 13/Output
//     PlcTask Outputs/.P10_050_DO1.PDOS.PlcToHw.digitalOutput_14 <-> Channel 14/Output
//     PlcTask Outputs/.P10_050_DO1.PDOS.PlcToHw.digitalOutput_15 <-> Channel 15/Output
//     PlcTask Outputs/.P10_050_DO1.PDOS.PlcToHw.digitalOutput_16 <-> Channel 16/Output
//   Plc_Prog/Plc_Prog Instance <-> ETH/+P10=050-BC1 - Press / Dryer PLC Cabinet/+P10=050-DO2 (EL2809)
//     PlcTask Outputs/.P10_050_DO2.PDOS.PlcToHw.digitalOutput_01 <-> Channel 1/Output
//     PlcTask Outputs/.P10_050_DO2.PDOS.PlcToHw.digitalOutput_02 <-> Channel 2/Output
//     PlcTask Outputs/.P10_050_DO2.PDOS.PlcToHw.digitalOutput_03 <-> Channel 3/Output
//     PlcTask Outputs/.P10_050_DO2.PDOS.PlcToHw.digitalOutput_04 <-> Channel 4/Output
//     PlcTask Outputs/.P10_050_DO2.PDOS.PlcToHw.digitalOutput_05 <-> Channel 5/Output
//     PlcTask Outputs/.P10_050_DO2.PDOS.PlcToHw.digitalOutput_06 <-> Channel 6/Output
//     PlcTask Outputs/.P10_050_DO2.PDOS.PlcToHw.digitalOutput_07 <-> Channel 7/Output
//     PlcTask Outputs/.P10_050_DO2.PDOS.PlcToHw.digitalOutput_08 <-> Channel 8/Output
//     PlcTask Outputs/.P10_050_DO2.PDOS.PlcToHw.digitalOutput_09 <-> Channel 9/Output
//     PlcTask Outputs/.P10_050_DO2.PDOS.PlcToHw.digitalOutput_10 <-> Channel 10/Output
//     PlcTask Outputs/.P10_050_DO2.PDOS.PlcToHw.digitalOutput_11 <-> Channel 11/Output
//     PlcTask Outputs/.P10_050_DO2.PDOS.PlcToHw.digitalOutput_12 <-> Channel 12/Output
//     PlcTask Outputs/.P10_050_DO2.PDOS.PlcToHw.digitalOutput_13 <-> Channel 13/Output
//     PlcTask Outputs/.P10_050_DO2.PDOS.PlcToHw.digitalOutput_14 <-> Channel 14/Output
//     PlcTask Outputs/.P10_050_DO2.PDOS.PlcToHw.digitalOutput_15 <-> Channel 15/Output
//     PlcTask Outputs/.P10_050_DO2.PDOS.PlcToHw.digitalOutput_16 <-> Channel 16/Output
//   Plc_Prog/Plc_Prog Instance <-> ETH/+P10=050-BC1 - Press / Dryer PLC Cabinet/+P10=050-DO3 (EL2809)
//     PlcTask Outputs/.P10_050_DO3.PDOS.PlcToHw.digitalOutput_01 <-> Channel 1/Output
//     PlcTask Outputs/.P10_050_DO3.PDOS.PlcToHw.digitalOutput_02 <-> Channel 2/Output
//     PlcTask Outputs/.P10_050_DO3.PDOS.PlcToHw.digitalOutput_03 <-> Channel 3/Output
//     PlcTask Outputs/.P10_050_DO3.PDOS.PlcToHw.digitalOutput_04 <-> Channel 4/Output
//     PlcTask Outputs/.P10_050_DO3.PDOS.PlcToHw.digitalOutput_05 <-> Channel 5/Output
//     PlcTask Outputs/.P10_050_DO3.PDOS.PlcToHw.digitalOutput_06 <-> Channel 6/Output
//     PlcTask Outputs/.P10_050_DO3.PDOS.PlcToHw.digitalOutput_07 <-> Channel 7/Output
//     PlcTask Outputs/.P10_050_DO3.PDOS.PlcToHw.digitalOutput_08 <-> Channel 8/Output
//     PlcTask Outputs/.P10_050_DO3.PDOS.PlcToHw.digitalOutput_09 <-> Channel 9/Output
//     PlcTask Outputs/.P10_050_DO3.PDOS.PlcToHw.digitalOutput_10 <-> Channel 10/Output
//     PlcTask Outputs/.P10_050_DO3.PDOS.PlcToHw.digitalOutput_11 <-> Channel 11/Output
//     PlcTask Outputs/.P10_050_DO3.PDOS.PlcToHw.digitalOutput_12 <-> Channel 12/Output
//     PlcTask Outputs/.P10_050_DO3.PDOS.PlcToHw.digitalOutput_13 <-> Channel 13/Output
//     PlcTask Outputs/.P10_050_DO3.PDOS.PlcToHw.digitalOutput_14 <-> Channel 14/Output
//     PlcTask Outputs/.P10_050_DO3.PDOS.PlcToHw.digitalOutput_15 <-> Channel 15/Output
//     PlcTask Outputs/.P10_050_DO3.PDOS.PlcToHw.digitalOutput_16 <-> Channel 16/Output
//   Plc_Prog/Plc_Prog Instance <-> ETH/+P10=050-BC1 - Press / Dryer PLC Cabinet/+P10=050-DO4 (EL2809)
//     PlcTask Outputs/.P10_050_DO4.PDOS.PlcToHw.digitalOutput_01 <-> Channel 1/Output
//     PlcTask Outputs/.P10_050_DO4.PDOS.PlcToHw.digitalOutput_02 <-> Channel 2/Output
//     PlcTask Outputs/.P10_050_DO4.PDOS.PlcToHw.digitalOutput_03 <-> Channel 3/Output
//     PlcTask Outputs/.P10_050_DO4.PDOS.PlcToHw.digitalOutput_04 <-> Channel 4/Output
//     PlcTask Outputs/.P10_050_DO4.PDOS.PlcToHw.digitalOutput_05 <-> Channel 5/Output
//     PlcTask Outputs/.P10_050_DO4.PDOS.PlcToHw.digitalOutput_08 <-> Channel 8/Output
//     PlcTask Outputs/.P10_050_DO4.PDOS.PlcToHw.digitalOutput_09 <-> Channel 9/Output
//     PlcTask Outputs/.P10_050_DO4.PDOS.PlcToHw.digitalOutput_10 <-> Channel 10/Output
//     PlcTask Outputs/.P10_050_DO4.PDOS.PlcToHw.digitalOutput_11 <-> Channel 11/Output
//     PlcTask Outputs/.P10_050_DO4.PDOS.PlcToHw.digitalOutput_12 <-> Channel 12/Output
//     PlcTask Outputs/.P10_050_DO4.PDOS.PlcToHw.digitalOutput_13 <-> Channel 13/Output
//     PlcTask Outputs/.P10_050_DO4.PDOS.PlcToHw.digitalOutput_14 <-> Channel 14/Output
//     PlcTask Outputs/.P10_050_DO4.PDOS.PlcToHw.digitalOutput_15 <-> Channel 15/Output
//     PlcTask Outputs/.P10_050_DO4.PDOS.PlcToHw.digitalOutput_16 <-> Channel 16/Output
//     PlcTask Outputs/.P10_050_DO4.PDOS.PlcToHw.digitalOutput_06 <-> Channel 6/.P10_050_DO4.PDOS.PlcToHw.digitalOutput_06
//     PlcTask Outputs/.P10_050_DO4.PDOS.PlcToHw.digitalOutput_07 <-> Channel 7/.P10_050_DO4.PDOS.PlcToHw.digitalOutput_07
//   Plc_Prog/Plc_Prog Instance <-> ETH/+P10=050-BC2 - Press / Dryer PLC Cabinet/+P10=050-AI1 (EL3054)
//     PlcTask Inputs/.P10_050_AI1.PDOS.HwToPLC.Channel1/Status/Overrange <-> AI Standard Channel 1/Status/Overrange
//     PlcTask Inputs/.P10_050_AI1.PDOS.HwToPLC.Channel2/Status/Overrange <-> AI Standard Channel 2/Status/Overrange
//     PlcTask Inputs/.P10_050_AI1.PDOS.HwToPLC.Channel3/Status/Overrange <-> AI Standard Channel 3/Status/Overrange
//     PlcTask Inputs/.P10_050_AI1.PDOS.HwToPLC.Channel4/Status/Overrange <-> AI Standard Channel 4/Status/Overrange
//     PlcTask Inputs/.P10_050_AI1.PDOS.HwToPLC.Channel1/Status/Underrange <-> AI Standard Channel 1/Status/Underrange
//     PlcTask Inputs/.P10_050_AI1.PDOS.HwToPLC.Channel2/Status/Underrange <-> AI Standard Channel 2/Status/Underrange
//     PlcTask Inputs/.P10_050_AI1.PDOS.HwToPLC.Channel3/Status/Underrange <-> AI Standard Channel 3/Status/Underrange
//     PlcTask Inputs/.P10_050_AI1.PDOS.HwToPLC.Channel4/Status/Underrange <-> AI Standard Channel 4/Status/Underrange
//     PlcTask Inputs/.P10_050_AI1.PDOS.HwToPLC.Channel1/Value <-> AI Standard Channel 1/Value
//     PlcTask Inputs/.P10_050_AI1.PDOS.HwToPLC.Channel2/Value <-> AI Standard Channel 2/Value
//     PlcTask Inputs/.P10_050_AI1.PDOS.HwToPLC.Channel3/Value <-> AI Standard Channel 3/Value
//     PlcTask Inputs/.P10_050_AI1.PDOS.HwToPLC.Channel4/Value <-> AI Standard Channel 4/Value
//   Plc_Prog/Plc_Prog Instance <-> ETH/+P10=050-BC2 - Press / Dryer PLC Cabinet/+P10=050-AI2 (EL3204)
//     PlcTask Inputs/.P10_050_AI2.PDOS.HwToPLC.Channel1/Status/Overrange <-> RTD Inputs Channel 1/Status/Overrange
//     PlcTask Inputs/.P10_050_AI2.PDOS.HwToPLC.Channel2/Status/Overrange <-> RTD Inputs Channel 2/Status/Overrange
//     PlcTask Inputs/.P10_050_AI2.PDOS.HwToPLC.Channel3/Status/Overrange <-> RTD Inputs Channel 4/Status/Overrange
//     PlcTask Inputs/.P10_050_AI2.PDOS.HwToPLC.Channel4/Status/Overrange <-> RTD Inputs Channel 3/Status/Overrange
//     PlcTask Inputs/.P10_050_AI2.PDOS.HwToPLC.Channel1/Status/Underrange <-> RTD Inputs Channel 1/Status/Underrange
//     PlcTask Inputs/.P10_050_AI2.PDOS.HwToPLC.Channel2/Status/Underrange <-> RTD Inputs Channel 2/Status/Underrange
//     PlcTask Inputs/.P10_050_AI2.PDOS.HwToPLC.Channel3/Status/Underrange <-> RTD Inputs Channel 4/Status/Underrange
//     PlcTask Inputs/.P10_050_AI2.PDOS.HwToPLC.Channel4/Status/Underrange <-> RTD Inputs Channel 3/Status/Underrange
//     PlcTask Inputs/.P10_050_AI2.PDOS.HwToPLC.Channel1/Value <-> RTD Inputs Channel 1/Value
//     PlcTask Inputs/.P10_050_AI2.PDOS.HwToPLC.Channel2/Value <-> RTD Inputs Channel 2/Value
//     PlcTask Inputs/.P10_050_AI2.PDOS.HwToPLC.Channel3/Value <-> RTD Inputs Channel 3/Value
//     PlcTask Inputs/.P10_050_AI2.PDOS.HwToPLC.Channel4/Value <-> RTD Inputs Channel 4/Value
//   Plc_Prog/Plc_Prog Instance <-> ETH/+P10=050-BC2 - Press / Dryer PLC Cabinet/+P10=050-AO1(EL4024)
//     PlcTask Outputs/.P10_050_AO1.PDOS.HwToPLC.Channel1 <-> AO Outputs Channel 1/Analog output
//     PlcTask Outputs/.P10_050_AO1.PDOS.HwToPLC.Channel2 <-> AO Outputs Channel 2/Analog output
//     PlcTask Outputs/.P10_050_AO1.PDOS.HwToPLC.Channel3 <-> AO Outputs Channel 3/Analog output
//     PlcTask Outputs/.P10_050_AO1.PDOS.HwToPLC.Channel4 <-> AO Outputs Channel 4/Analog output
//   Plc_Prog/Plc_Prog Instance <-> ETH/+P11=400-UG1 - Second Press
//     PlcTask Inputs/.P11_400_UG01_SecondPress.PDOS.DrvToPLC.errorCode <-> 1st TxPDO Mapping/Error code
//     PlcTask Inputs/.P11_400_UG01_SecondPress.PDOS.DrvToPLC.modesOfOperationDisplay <-> 1st TxPDO Mapping/Mode Of Operation Display
//     PlcTask Inputs/.P11_400_UG01_SecondPress.PDOS.DrvToPLC.positionActualValue <-> 1st TxPDO Mapping/Position actual value
//     PlcTask Inputs/.P11_400_UG01_SecondPress.PDOS.DrvToPLC.statusWord <-> 1st TxPDO Mapping/Status Word
//     PlcTask Inputs/.P11_400_UG01_SecondPress.PDOS.DrvToPLC.torqueActualValue <-> 1st TxPDO Mapping/Torque actual value
//     PlcTask Inputs/.P11_400_UG01_SecondPress.PDOS.DrvToPLC.velocityActualValue <-> 1st TxPDO Mapping/Velocity actual value
//     PlcTask Outputs/.P11_400_UG01_SecondPress.PDOS.PlcToDrv.controlWord <-> 1st RxPDO Mapping/Control Word
//     PlcTask Outputs/.P11_400_UG01_SecondPress.PDOS.PlcToDrv.maxMotorSpeed <-> 1st RxPDO Mapping/Max motor speed
//     PlcTask Outputs/.P11_400_UG01_SecondPress.PDOS.PlcToDrv.maxTorque <-> 1st RxPDO Mapping/Target torque
//     PlcTask Outputs/.P11_400_UG01_SecondPress.PDOS.PlcToDrv.modesOfOperation <-> 1st RxPDO Mapping/Modes of operation
//     PlcTask Outputs/.P11_400_UG01_SecondPress.PDOS.PlcToDrv.vlTargetVelocity <-> 1st RxPDO Mapping/vl target velocity
//   Plc_Prog/Plc_Prog Instance <-> ETH/+P12=400-UG1 - First Press
//     PlcTask Inputs/.P12_400_UG01_FirstPress.PDOS.DrvToPLC.errorCode <-> 1st TxPDO Mapping/Error code
//     PlcTask Inputs/.P12_400_UG01_FirstPress.PDOS.DrvToPLC.modesOfOperationDisplay <-> 1st TxPDO Mapping/Mode Of Operation Display
//     PlcTask Inputs/.P12_400_UG01_FirstPress.PDOS.DrvToPLC.positionActualValue <-> 1st TxPDO Mapping/Position actual value
//     PlcTask Inputs/.P12_400_UG01_FirstPress.PDOS.DrvToPLC.statusWord <-> 1st TxPDO Mapping/Status Word
//     PlcTask Inputs/.P12_400_UG01_FirstPress.PDOS.DrvToPLC.torqueActualValue <-> 1st TxPDO Mapping/Torque actual value
//     PlcTask Inputs/.P12_400_UG01_FirstPress.PDOS.DrvToPLC.velocityActualValue <-> 1st TxPDO Mapping/Velocity actual value
//     PlcTask Outputs/.P12_400_UG01_FirstPress.PDOS.PlcToDrv.controlWord <-> 1st RxPDO Mapping/Control Word
//     PlcTask Outputs/.P12_400_UG01_FirstPress.PDOS.PlcToDrv.maxMotorSpeed <-> 1st RxPDO Mapping/Max motor speed
//     PlcTask Outputs/.P12_400_UG01_FirstPress.PDOS.PlcToDrv.maxTorque <-> 1st RxPDO Mapping/Target torque
//     PlcTask Outputs/.P12_400_UG01_FirstPress.PDOS.PlcToDrv.modesOfOperation <-> 1st RxPDO Mapping/Modes of operation
//     PlcTask Outputs/.P12_400_UG01_FirstPress.PDOS.PlcToDrv.vlTargetVelocity <-> 1st RxPDO Mapping/vl target velocity
//   Plc_Prog/Plc_Prog Instance <-> ETH/+P12=500-UG2 - Dryer Section GR1 - Lower GR1 Master
//     PlcTask Inputs/.P13_500_UG02_1GR_LowerMaster.PDOS.DrvToPLC.errorCode <-> 1st TxPDO Mapping/Error code
//     PlcTask Inputs/.P13_500_UG02_1GR_LowerMaster.PDOS.DrvToPLC.modesOfOperationDisplay <-> 1st TxPDO Mapping/Mode Of Operation Display
//     PlcTask Inputs/.P13_500_UG02_1GR_LowerMaster.PDOS.DrvToPLC.positionActualValue <-> 1st TxPDO Mapping/Position actual value
//     PlcTask Inputs/.P13_500_UG02_1GR_LowerMaster.PDOS.DrvToPLC.statusWord <-> 1st TxPDO Mapping/Status Word
//     PlcTask Inputs/.P13_500_UG02_1GR_LowerMaster.PDOS.DrvToPLC.torqueActualValue <-> 1st TxPDO Mapping/Torque actual value
//     PlcTask Inputs/.P13_500_UG02_1GR_LowerMaster.PDOS.DrvToPLC.velocityActualValue <-> 1st TxPDO Mapping/Velocity actual value
//     PlcTask Outputs/.P13_500_UG02_1GR_LowerMaster.PDOS.PlcToDrv.controlWord <-> 1st RxPDO Mapping/Control Word
//     PlcTask Outputs/.P13_500_UG02_1GR_LowerMaster.PDOS.PlcToDrv.maxMotorSpeed <-> 1st RxPDO Mapping/Max motor speed
//     PlcTask Outputs/.P13_500_UG02_1GR_LowerMaster.PDOS.PlcToDrv.maxTorque <-> 1st RxPDO Mapping/Target torque
//     PlcTask Outputs/.P13_500_UG02_1GR_LowerMaster.PDOS.PlcToDrv.modesOfOperation <-> 1st RxPDO Mapping/Modes of operation
//     PlcTask Outputs/.P13_500_UG02_1GR_LowerMaster.PDOS.PlcToDrv.vlTargetVelocity <-> 1st RxPDO Mapping/vl target velocity
//   Plc_Prog/Plc_Prog Instance <-> ETH/+P12=500-UG3 - Dryer Section GR1 - Upper Master
//     PlcTask Inputs/.P13_500_UG03_1GR_UpperMaster.PDOS.DrvToPLC.errorCode <-> 1st TxPDO Mapping/Error code
//     PlcTask Inputs/.P13_500_UG03_1GR_UpperMaster.PDOS.DrvToPLC.modesOfOperationDisplay <-> 1st TxPDO Mapping/Mode Of Operation Display
//     PlcTask Inputs/.P13_500_UG03_1GR_UpperMaster.PDOS.DrvToPLC.positionActualValue <-> 1st TxPDO Mapping/Position actual value
//     PlcTask Inputs/.P13_500_UG03_1GR_UpperMaster.PDOS.DrvToPLC.statusWord <-> 1st TxPDO Mapping/Status Word
//     PlcTask Inputs/.P13_500_UG03_1GR_UpperMaster.PDOS.DrvToPLC.torqueActualValue <-> 1st TxPDO Mapping/Torque actual value
//     PlcTask Inputs/.P13_500_UG03_1GR_UpperMaster.PDOS.DrvToPLC.velocityActualValue <-> 1st TxPDO Mapping/Velocity actual value
//     PlcTask Outputs/.P13_500_UG03_1GR_UpperMaster.PDOS.PlcToDrv.controlWord <-> 1st RxPDO Mapping/Control Word
//     PlcTask Outputs/.P13_500_UG03_1GR_UpperMaster.PDOS.PlcToDrv.maxMotorSpeed <-> 1st RxPDO Mapping/Max motor speed
//     PlcTask Outputs/.P13_500_UG03_1GR_UpperMaster.PDOS.PlcToDrv.maxTorque <-> 1st RxPDO Mapping/Target torque
//     PlcTask Outputs/.P13_500_UG03_1GR_UpperMaster.PDOS.PlcToDrv.modesOfOperation <-> 1st RxPDO Mapping/Modes of operation
//     PlcTask Outputs/.P13_500_UG03_1GR_UpperMaster.PDOS.PlcToDrv.vlTargetVelocity <-> 1st RxPDO Mapping/vl target velocity
//   Plc_Prog/Plc_Prog Instance <-> ETH/+P12=501-UG1 - Dryer Section  GR2 - Lower Slave
//     PlcTask Inputs/.P13_501_UG01_2GR_LowerSlave.PDOS.DrvToPLC.errorCode <-> 1st TxPDO Mapping/Error code
//     PlcTask Inputs/.P13_501_UG01_2GR_LowerSlave.PDOS.DrvToPLC.modesOfOperationDisplay <-> 1st TxPDO Mapping/Mode Of Operation Display
//     PlcTask Inputs/.P13_501_UG01_2GR_LowerSlave.PDOS.DrvToPLC.positionActualValue <-> 1st TxPDO Mapping/Position actual value
//     PlcTask Inputs/.P13_501_UG01_2GR_LowerSlave.PDOS.DrvToPLC.statusWord <-> 1st TxPDO Mapping/Status Word
//     PlcTask Inputs/.P13_501_UG01_2GR_LowerSlave.PDOS.DrvToPLC.torqueActualValue <-> 1st TxPDO Mapping/Torque actual value
//     PlcTask Inputs/.P13_501_UG01_2GR_LowerSlave.PDOS.DrvToPLC.velocityActualValue <-> 1st TxPDO Mapping/Velocity actual value
//     PlcTask Outputs/.P13_501_UG01_2GR_LowerSlave.PDOS.PlcToDrv.controlWord <-> 1st RxPDO Mapping/Control Word
//     PlcTask Outputs/.P13_501_UG01_2GR_LowerSlave.PDOS.PlcToDrv.maxMotorSpeed <-> 1st RxPDO Mapping/Max motor speed
//     PlcTask Outputs/.P13_501_UG01_2GR_LowerSlave.PDOS.PlcToDrv.maxTorque <-> 1st RxPDO Mapping/Target torque
//     PlcTask Outputs/.P13_501_UG01_2GR_LowerSlave.PDOS.PlcToDrv.modesOfOperation <-> 1st RxPDO Mapping/Modes of operation
//     PlcTask Outputs/.P13_501_UG01_2GR_LowerSlave.PDOS.PlcToDrv.vlTargetVelocity <-> 1st RxPDO Mapping/vl target velocity
//   Plc_Prog/Plc_Prog Instance <-> ETH/+P12=501-UG2 - Dryer Section GR2 - Upper Slave
//     PlcTask Inputs/.P13_501_UG02_2GR_UpperSlave.PDOS.DrvToPLC.errorCode <-> 1st TxPDO Mapping/Error code
//     PlcTask Inputs/.P13_501_UG02_2GR_UpperSlave.PDOS.DrvToPLC.modesOfOperationDisplay <-> 1st TxPDO Mapping/Mode Of Operation Display
//     PlcTask Inputs/.P13_501_UG02_2GR_UpperSlave.PDOS.DrvToPLC.positionActualValue <-> 1st TxPDO Mapping/Position actual value
//     PlcTask Inputs/.P13_501_UG02_2GR_UpperSlave.PDOS.DrvToPLC.statusWord <-> 1st TxPDO Mapping/Status Word
//     PlcTask Inputs/.P13_501_UG02_2GR_UpperSlave.PDOS.DrvToPLC.torqueActualValue <-> 1st TxPDO Mapping/Torque actual value
//     PlcTask Inputs/.P13_501_UG02_2GR_UpperSlave.PDOS.DrvToPLC.velocityActualValue <-> 1st TxPDO Mapping/Velocity actual value
//     PlcTask Outputs/.P13_501_UG02_2GR_UpperSlave.PDOS.PlcToDrv.controlWord <-> 1st RxPDO Mapping/Control Word
//     PlcTask Outputs/.P13_501_UG02_2GR_UpperSlave.PDOS.PlcToDrv.maxMotorSpeed <-> 1st RxPDO Mapping/Max motor speed
//     PlcTask Outputs/.P13_501_UG02_2GR_UpperSlave.PDOS.PlcToDrv.maxTorque <-> 1st RxPDO Mapping/Target torque
//     PlcTask Outputs/.P13_501_UG02_2GR_UpperSlave.PDOS.PlcToDrv.modesOfOperation <-> 1st RxPDO Mapping/Modes of operation
//     PlcTask Outputs/.P13_501_UG02_2GR_UpperSlave.PDOS.PlcToDrv.vlTargetVelocity <-> 1st RxPDO Mapping/vl target velocity
//   Plc_Prog/Plc_Prog Instance <-> ETH/+P12=501-UG3 - Dryer Section GR2 - Lower Master
//     PlcTask Inputs/.P13_501_UG03_2GR_LowerMaster.PDOS.DrvToPLC.errorCode <-> 1st TxPDO Mapping/Error code
//     PlcTask Inputs/.P13_501_UG03_2GR_LowerMaster.PDOS.DrvToPLC.modesOfOperationDisplay <-> 1st TxPDO Mapping/Mode Of Operation Display
//     PlcTask Inputs/.P13_501_UG03_2GR_LowerMaster.PDOS.DrvToPLC.positionActualValue <-> 1st TxPDO Mapping/Position actual value
//     PlcTask Inputs/.P13_501_UG03_2GR_LowerMaster.PDOS.DrvToPLC.statusWord <-> 1st TxPDO Mapping/Status Word
//     PlcTask Inputs/.P13_501_UG03_2GR_LowerMaster.PDOS.DrvToPLC.torqueActualValue <-> 1st TxPDO Mapping/Torque actual value
//     PlcTask Inputs/.P13_501_UG03_2GR_LowerMaster.PDOS.DrvToPLC.velocityActualValue <-> 1st TxPDO Mapping/Velocity actual value
//     PlcTask Outputs/.P13_501_UG03_2GR_LowerMaster.PDOS.PlcToDrv.controlWord <-> 1st RxPDO Mapping/Control Word
//     PlcTask Outputs/.P13_501_UG03_2GR_LowerMaster.PDOS.PlcToDrv.maxMotorSpeed <-> 1st RxPDO Mapping/Max motor speed
//     PlcTask Outputs/.P13_501_UG03_2GR_LowerMaster.PDOS.PlcToDrv.maxTorque <-> 1st RxPDO Mapping/Target torque
//     PlcTask Outputs/.P13_501_UG03_2GR_LowerMaster.PDOS.PlcToDrv.modesOfOperation <-> 1st RxPDO Mapping/Modes of operation
//     PlcTask Outputs/.P13_501_UG03_2GR_LowerMaster.PDOS.PlcToDrv.vlTargetVelocity <-> 1st RxPDO Mapping/vl target velocity
//   Plc_Prog/Plc_Prog Instance <-> ETH/+P13=500-UG1 - Dryer Section GR1 - Upper GR1 Slave
//     PlcTask Inputs/.P13_500_UG01_1GR_UpperSlave.PDOS.DrvToPLC.errorCode <-> 1st TxPDO Mapping/Error code
//     PlcTask Inputs/.P13_500_UG01_1GR_UpperSlave.PDOS.DrvToPLC.modesOfOperationDisplay <-> 1st TxPDO Mapping/Mode Of Operation Display
//     PlcTask Inputs/.P13_500_UG01_1GR_UpperSlave.PDOS.DrvToPLC.positionActualValue <-> 1st TxPDO Mapping/Position actual value
//     PlcTask Inputs/.P13_500_UG01_1GR_UpperSlave.PDOS.DrvToPLC.statusWord <-> 1st TxPDO Mapping/Status Word
//     PlcTask Inputs/.P13_500_UG01_1GR_UpperSlave.PDOS.DrvToPLC.torqueActualValue <-> 1st TxPDO Mapping/Torque actual value
//     PlcTask Inputs/.P13_500_UG01_1GR_UpperSlave.PDOS.DrvToPLC.velocityActualValue <-> 1st TxPDO Mapping/Velocity actual value
//     PlcTask Outputs/.P13_500_UG01_1GR_UpperSlave.PDOS.PlcToDrv.controlWord <-> 1st RxPDO Mapping/Control Word
//     PlcTask Outputs/.P13_500_UG01_1GR_UpperSlave.PDOS.PlcToDrv.maxMotorSpeed <-> 1st RxPDO Mapping/Max motor speed
//     PlcTask Outputs/.P13_500_UG01_1GR_UpperSlave.PDOS.PlcToDrv.maxTorque <-> 1st RxPDO Mapping/Target torque
//     PlcTask Outputs/.P13_500_UG01_1GR_UpperSlave.PDOS.PlcToDrv.modesOfOperation <-> 1st RxPDO Mapping/Modes of operation
//     PlcTask Outputs/.P13_500_UG01_1GR_UpperSlave.PDOS.PlcToDrv.vlTargetVelocity <-> 1st RxPDO Mapping/vl target velocity
//   Plc_Prog/Plc_Prog Instance <-> ETH/+P13=501-UG1 - Dryer Section GR2 - Upper Master
//     PlcTask Inputs/.P14_501_UG01_2GR_UpperMaster.PDOS.DrvToPLC.errorCode <-> 1st TxPDO Mapping/Error code
//     PlcTask Inputs/.P14_501_UG01_2GR_UpperMaster.PDOS.DrvToPLC.modesOfOperationDisplay <-> 1st TxPDO Mapping/Mode Of Operation Display
//     PlcTask Inputs/.P14_501_UG01_2GR_UpperMaster.PDOS.DrvToPLC.positionActualValue <-> 1st TxPDO Mapping/Position actual value
//     PlcTask Inputs/.P14_501_UG01_2GR_UpperMaster.PDOS.DrvToPLC.statusWord <-> 1st TxPDO Mapping/Status Word
//     PlcTask Inputs/.P14_501_UG01_2GR_UpperMaster.PDOS.DrvToPLC.torqueActualValue <-> 1st TxPDO Mapping/Torque actual value
//     PlcTask Inputs/.P14_501_UG01_2GR_UpperMaster.PDOS.DrvToPLC.velocityActualValue <-> 1st TxPDO Mapping/Velocity actual value
//     PlcTask Outputs/.P14_501_UG01_2GR_UpperMaster.PDOS.PlcToDrv.controlWord <-> 1st RxPDO Mapping/Control Word
//     PlcTask Outputs/.P14_501_UG01_2GR_UpperMaster.PDOS.PlcToDrv.maxMotorSpeed <-> 1st RxPDO Mapping/Max motor speed
//     PlcTask Outputs/.P14_501_UG01_2GR_UpperMaster.PDOS.PlcToDrv.maxTorque <-> 1st RxPDO Mapping/Target torque
//     PlcTask Outputs/.P14_501_UG01_2GR_UpperMaster.PDOS.PlcToDrv.modesOfOperation <-> 1st RxPDO Mapping/Modes of operation
//     PlcTask Outputs/.P14_501_UG01_2GR_UpperMaster.PDOS.PlcToDrv.vlTargetVelocity <-> 1st RxPDO Mapping/vl target velocity
//   Plc_Prog/Plc_Prog Instance <-> ETH/+P13=502-UG2 - Dryer Section GR3 - Lower Slave
//     PlcTask Inputs/.P14_502_UG01_3GR_LowerSlave.PDOS.DrvToPLC.errorCode <-> 1st TxPDO Mapping/Error code
//     PlcTask Inputs/.P14_502_UG01_3GR_LowerSlave.PDOS.DrvToPLC.modesOfOperationDisplay <-> 1st TxPDO Mapping/Mode Of Operation Display
//     PlcTask Inputs/.P14_502_UG01_3GR_LowerSlave.PDOS.DrvToPLC.positionActualValue <-> 1st TxPDO Mapping/Position actual value
//     PlcTask Inputs/.P14_502_UG01_3GR_LowerSlave.PDOS.DrvToPLC.statusWord <-> 1st TxPDO Mapping/Status Word
//     PlcTask Inputs/.P14_502_UG01_3GR_LowerSlave.PDOS.DrvToPLC.torqueActualValue <-> 1st TxPDO Mapping/Torque actual value
//     PlcTask Inputs/.P14_502_UG01_3GR_LowerSlave.PDOS.DrvToPLC.velocityActualValue <-> 1st TxPDO Mapping/Velocity actual value
//     PlcTask Outputs/.P14_502_UG01_3GR_LowerSlave.PDOS.PlcToDrv.controlWord <-> 1st RxPDO Mapping/Control Word
//     PlcTask Outputs/.P14_502_UG01_3GR_LowerSlave.PDOS.PlcToDrv.maxMotorSpeed <-> 1st RxPDO Mapping/Max motor speed
//     PlcTask Outputs/.P14_502_UG01_3GR_LowerSlave.PDOS.PlcToDrv.maxTorque <-> 1st RxPDO Mapping/Target torque
//     PlcTask Outputs/.P14_502_UG01_3GR_LowerSlave.PDOS.PlcToDrv.modesOfOperation <-> 1st RxPDO Mapping/Modes of operation
//     PlcTask Outputs/.P14_502_UG01_3GR_LowerSlave.PDOS.PlcToDrv.vlTargetVelocity <-> 1st RxPDO Mapping/vl target velocity
//   Plc_Prog/Plc_Prog Instance <-> ETH/+P13=502-UG2 - Dryer Section GR3 - Upper Slave
//     PlcTask Inputs/.P14_502_UG02_3GR_UpperSlave.PDOS.DrvToPLC.errorCode <-> 1st TxPDO Mapping/Error code
//     PlcTask Inputs/.P14_502_UG02_3GR_UpperSlave.PDOS.DrvToPLC.modesOfOperationDisplay <-> 1st TxPDO Mapping/Mode Of Operation Display
//     PlcTask Inputs/.P14_502_UG02_3GR_UpperSlave.PDOS.DrvToPLC.positionActualValue <-> 1st TxPDO Mapping/Position actual value
//     PlcTask Inputs/.P14_502_UG02_3GR_UpperSlave.PDOS.DrvToPLC.statusWord <-> 1st TxPDO Mapping/Status Word
//     PlcTask Inputs/.P14_502_UG02_3GR_UpperSlave.PDOS.DrvToPLC.torqueActualValue <-> 1st TxPDO Mapping/Torque actual value
//     PlcTask Inputs/.P14_502_UG02_3GR_UpperSlave.PDOS.DrvToPLC.velocityActualValue <-> 1st TxPDO Mapping/Velocity actual value
//     PlcTask Outputs/.P14_502_UG02_3GR_UpperSlave.PDOS.PlcToDrv.controlWord <-> 1st RxPDO Mapping/Control Word
//     PlcTask Outputs/.P14_502_UG02_3GR_UpperSlave.PDOS.PlcToDrv.maxMotorSpeed <-> 1st RxPDO Mapping/Max motor speed
//     PlcTask Outputs/.P14_502_UG02_3GR_UpperSlave.PDOS.PlcToDrv.maxTorque <-> 1st RxPDO Mapping/Target torque
//     PlcTask Outputs/.P14_502_UG02_3GR_UpperSlave.PDOS.PlcToDrv.modesOfOperation <-> 1st RxPDO Mapping/Modes of operation
//     PlcTask Outputs/.P14_502_UG02_3GR_UpperSlave.PDOS.PlcToDrv.vlTargetVelocity <-> 1st RxPDO Mapping/vl target velocity
//   Plc_Prog/Plc_Prog Instance <-> ETH/+P13=502-UG3 - Dryer Section GR3 - Lower Master
//     PlcTask Inputs/.P14_502_UG03_3GR_LowerMaster.PDOS.DrvToPLC.errorCode <-> 1st TxPDO Mapping/Error code
//     PlcTask Inputs/.P14_502_UG03_3GR_LowerMaster.PDOS.DrvToPLC.modesOfOperationDisplay <-> 1st TxPDO Mapping/Mode Of Operation Display
//     PlcTask Inputs/.P14_502_UG03_3GR_LowerMaster.PDOS.DrvToPLC.positionActualValue <-> 1st TxPDO Mapping/Position actual value
//     PlcTask Inputs/.P14_502_UG03_3GR_LowerMaster.PDOS.DrvToPLC.statusWord <-> 1st TxPDO Mapping/Status Word
//     PlcTask Inputs/.P14_502_UG03_3GR_LowerMaster.PDOS.DrvToPLC.torqueActualValue <-> 1st TxPDO Mapping/Torque actual value
//     PlcTask Inputs/.P14_502_UG03_3GR_LowerMaster.PDOS.DrvToPLC.velocityActualValue <-> 1st TxPDO Mapping/Velocity actual value
//     PlcTask Outputs/.P14_502_UG03_3GR_LowerMaster.PDOS.PlcToDrv.controlWord <-> 1st RxPDO Mapping/Control Word
//     PlcTask Outputs/.P14_502_UG03_3GR_LowerMaster.PDOS.PlcToDrv.maxMotorSpeed <-> 1st RxPDO Mapping/Max motor speed
//     PlcTask Outputs/.P14_502_UG03_3GR_LowerMaster.PDOS.PlcToDrv.maxTorque <-> 1st RxPDO Mapping/Target torque
//     PlcTask Outputs/.P14_502_UG03_3GR_LowerMaster.PDOS.PlcToDrv.modesOfOperation <-> 1st RxPDO Mapping/Modes of operation
//     PlcTask Outputs/.P14_502_UG03_3GR_LowerMaster.PDOS.PlcToDrv.vlTargetVelocity <-> 1st RxPDO Mapping/vl target velocity
//   Plc_Prog/Plc_Prog Instance <-> ETH/+P13=502-UG4 - Dryer Section GR3 - Upper Master
//     PlcTask Inputs/.P14_502_UG04_3GR_UpperMaster.PDOS.DrvToPLC.errorCode <-> 1st TxPDO Mapping/Error code
//     PlcTask Inputs/.P14_502_UG04_3GR_UpperMaster.PDOS.DrvToPLC.modesOfOperationDisplay <-> 1st TxPDO Mapping/Mode Of Operation Display
//     PlcTask Inputs/.P14_502_UG04_3GR_UpperMaster.PDOS.DrvToPLC.positionActualValue <-> 1st TxPDO Mapping/Position actual value
//     PlcTask Inputs/.P14_502_UG04_3GR_UpperMaster.PDOS.DrvToPLC.statusWord <-> 1st TxPDO Mapping/Status Word
//     PlcTask Inputs/.P14_502_UG04_3GR_UpperMaster.PDOS.DrvToPLC.torqueActualValue <-> 1st TxPDO Mapping/Torque actual value
//     PlcTask Inputs/.P14_502_UG04_3GR_UpperMaster.PDOS.DrvToPLC.velocityActualValue <-> 1st TxPDO Mapping/Velocity actual value
//     PlcTask Outputs/.P14_502_UG04_3GR_UpperMaster.PDOS.PlcToDrv.controlWord <-> 1st RxPDO Mapping/Control Word
//     PlcTask Outputs/.P14_502_UG04_3GR_UpperMaster.PDOS.PlcToDrv.maxMotorSpeed <-> 1st RxPDO Mapping/Max motor speed
//     PlcTask Outputs/.P14_502_UG04_3GR_UpperMaster.PDOS.PlcToDrv.maxTorque <-> 1st RxPDO Mapping/Target torque
//     PlcTask Outputs/.P14_502_UG04_3GR_UpperMaster.PDOS.PlcToDrv.modesOfOperation <-> 1st RxPDO Mapping/Modes of operation
//     PlcTask Outputs/.P14_502_UG04_3GR_UpperMaster.PDOS.PlcToDrv.vlTargetVelocity <-> 1st RxPDO Mapping/vl target velocity
//   Plc_Prog/Plc_Prog Instance <-> ETH/+P14=600-UG1 - Winder
//     PlcTask Inputs/.P15_600_UG01_Rewinder.PDOS.DrvToPLC.errorCode <-> 1st TxPDO Mapping/Error code
//     PlcTask Inputs/.P15_600_UG01_Rewinder.PDOS.DrvToPLC.modesOfOperationDisplay <-> 1st TxPDO Mapping/Mode Of Operation Display
//     PlcTask Inputs/.P15_600_UG01_Rewinder.PDOS.DrvToPLC.positionActualValue <-> 1st TxPDO Mapping/Position actual value
//     PlcTask Inputs/.P15_600_UG01_Rewinder.PDOS.DrvToPLC.statusWord <-> 1st TxPDO Mapping/Status Word
//     PlcTask Inputs/.P15_600_UG01_Rewinder.PDOS.DrvToPLC.torqueActualValue <-> 1st TxPDO Mapping/Torque actual value
//     PlcTask Inputs/.P15_600_UG01_Rewinder.PDOS.DrvToPLC.velocityActualValue <-> 1st TxPDO Mapping/Velocity actual value
//     PlcTask Outputs/.P15_600_UG01_Rewinder.PDOS.PlcToDrv.controlWord <-> 1st RxPDO Mapping/Control Word
//     PlcTask Outputs/.P15_600_UG01_Rewinder.PDOS.PlcToDrv.maxMotorSpeed <-> 1st RxPDO Mapping/Max motor speed
//     PlcTask Outputs/.P15_600_UG01_Rewinder.PDOS.PlcToDrv.maxTorque <-> 1st RxPDO Mapping/Target torque
//     PlcTask Outputs/.P15_600_UG01_Rewinder.PDOS.PlcToDrv.modesOfOperation <-> 1st RxPDO Mapping/Modes of operation
//     PlcTask Outputs/.P15_600_UG01_Rewinder.PDOS.PlcToDrv.vlTargetVelocity <-> 1st RxPDO Mapping/vl target velocity
//   Plc_Prog/Plc_Prog Instance <-> ETH/+P2=100-UG1 - Drive Roll
//     PlcTask Inputs/.P1_300_UG06_TractionRoll.PDOS.DrvToPLC.errorCode <-> 1st TxPDO Mapping/Error code
//     PlcTask Inputs/.P1_300_UG06_TractionRoll.PDOS.DrvToPLC.modesOfOperationDisplay <-> 1st TxPDO Mapping/Mode Of Operation Display
//     PlcTask Inputs/.P1_300_UG06_TractionRoll.PDOS.DrvToPLC.positionActualValue <-> 1st TxPDO Mapping/Position actual value
//     PlcTask Inputs/.P1_300_UG06_TractionRoll.PDOS.DrvToPLC.statusWord <-> 1st TxPDO Mapping/Status Word
//     PlcTask Inputs/.P1_300_UG06_TractionRoll.PDOS.DrvToPLC.torqueActualValue <-> 1st TxPDO Mapping/Torque actual value
//     PlcTask Inputs/.P1_300_UG06_TractionRoll.PDOS.DrvToPLC.velocityActualValue <-> 1st TxPDO Mapping/Velocity actual value
//     PlcTask Outputs/.P1_300_UG06_TractionRoll.PDOS.PlcToDrv.controlWord <-> 1st RxPDO Mapping/Control Word
//     PlcTask Outputs/.P1_300_UG06_TractionRoll.PDOS.PlcToDrv.maxMotorSpeed <-> 1st RxPDO Mapping/Max motor speed
//     PlcTask Outputs/.P1_300_UG06_TractionRoll.PDOS.PlcToDrv.maxTorque <-> 1st RxPDO Mapping/Max torque
//     PlcTask Outputs/.P1_300_UG06_TractionRoll.PDOS.PlcToDrv.modesOfOperation <-> 1st RxPDO Mapping/Modes of operation
//     PlcTask Outputs/.P1_300_UG06_TractionRoll.PDOS.PlcToDrv.vlTargetVelocity <-> 1st RxPDO Mapping/vl target velocity
//   Plc_Prog/Plc_Prog Instance <-> ETH/+P3=100-UG1 - CouchPit
//     PlcTask Inputs/.P1_100_UG04.PDOS.DrvToPLC.errorCode <-> 1st TxPDO Mapping/Error code
//     PlcTask Inputs/.P1_100_UG04.PDOS.DrvToPLC.modesOfOperationDisplay <-> 1st TxPDO Mapping/Mode Of Operation Display
//     PlcTask Inputs/.P1_100_UG04.PDOS.DrvToPLC.positionActualValue <-> 1st TxPDO Mapping/Position actual value
//     PlcTask Inputs/.P1_100_UG04.PDOS.DrvToPLC.statusWord <-> 1st TxPDO Mapping/Status Word
//     PlcTask Inputs/.P1_100_UG04.PDOS.DrvToPLC.torqueActualValue <-> 1st TxPDO Mapping/Torque actual value
//     PlcTask Inputs/.P1_100_UG04.PDOS.DrvToPLC.velocityActualValue <-> 1st TxPDO Mapping/Velocity actual value
//     PlcTask Outputs/.P1_100_UG04.PDOS.PlcToDrv.controlWord <-> 1st RxPDO Mapping/Control Word
//     PlcTask Outputs/.P1_100_UG04.PDOS.PlcToDrv.maxMotorSpeed <-> 1st RxPDO Mapping/Max motor speed
//     PlcTask Outputs/.P1_100_UG04.PDOS.PlcToDrv.maxTorque <-> 1st RxPDO Mapping/Max torque
//     PlcTask Outputs/.P1_100_UG04.PDOS.PlcToDrv.modesOfOperation <-> 1st RxPDO Mapping/Modes of operation
//     PlcTask Outputs/.P1_100_UG04.PDOS.PlcToDrv.vlTargetVelocity <-> 1st RxPDO Mapping/vl target velocity
//   Plc_Prog/Plc_Prog Instance <-> ETH/+P3=100-UG1 - SuctionRoll
//     PlcTask Inputs/.P1_100_UG03_SuctionRoll.PDOS.DrvToPLC.errorCode <-> 1st TxPDO Mapping/Error code
//     PlcTask Inputs/.P1_100_UG03_SuctionRoll.PDOS.DrvToPLC.modesOfOperationDisplay <-> 1st TxPDO Mapping/Mode Of Operation Display
//     PlcTask Inputs/.P1_100_UG03_SuctionRoll.PDOS.DrvToPLC.positionActualValue <-> 1st TxPDO Mapping/Position actual value
//     PlcTask Inputs/.P1_100_UG03_SuctionRoll.PDOS.DrvToPLC.statusWord <-> 1st TxPDO Mapping/Status Word
//     PlcTask Inputs/.P1_100_UG03_SuctionRoll.PDOS.DrvToPLC.torqueActualValue <-> 1st TxPDO Mapping/Torque actual value
//     PlcTask Inputs/.P1_100_UG03_SuctionRoll.PDOS.DrvToPLC.velocityActualValue <-> 1st TxPDO Mapping/Velocity actual value
//     PlcTask Outputs/.P1_100_UG03_SuctionRoll.PDOS.PlcToDrv.controlWord <-> 1st RxPDO Mapping/Control Word
//     PlcTask Outputs/.P1_100_UG03_SuctionRoll.PDOS.PlcToDrv.maxMotorSpeed <-> 1st RxPDO Mapping/Max motor speed
//     PlcTask Outputs/.P1_100_UG03_SuctionRoll.PDOS.PlcToDrv.maxTorque <-> 1st RxPDO Mapping/Target torque
//     PlcTask Outputs/.P1_100_UG03_SuctionRoll.PDOS.PlcToDrv.modesOfOperation <-> 1st RxPDO Mapping/Modes of operation
//     PlcTask Outputs/.P1_100_UG03_SuctionRoll.PDOS.PlcToDrv.vlTargetVelocity <-> 1st RxPDO Mapping/vl target velocity
//   Plc_Prog/Plc_Prog Instance <-> ETH/+P3=100-UG2 - Stock pump
//     PlcTask Inputs/.P1_100_UG05.PDOS.DrvToPLC.errorCode <-> 1st TxPDO Mapping/Error code
//     PlcTask Inputs/.P1_100_UG05.PDOS.DrvToPLC.modesOfOperationDisplay <-> 1st TxPDO Mapping/Mode Of Operation Display
//     PlcTask Inputs/.P1_100_UG05.PDOS.DrvToPLC.positionActualValue <-> 1st TxPDO Mapping/Position actual value
//     PlcTask Inputs/.P1_100_UG05.PDOS.DrvToPLC.statusWord <-> 1st TxPDO Mapping/Status Word
//     PlcTask Inputs/.P1_100_UG05.PDOS.DrvToPLC.torqueActualValue <-> 1st TxPDO Mapping/Torque actual value
//     PlcTask Inputs/.P1_100_UG05.PDOS.DrvToPLC.velocityActualValue <-> 1st TxPDO Mapping/Velocity actual value
//     PlcTask Outputs/.P1_100_UG05.PDOS.PlcToDrv.controlWord <-> 1st RxPDO Mapping/Control Word
//     PlcTask Outputs/.P1_100_UG05.PDOS.PlcToDrv.maxMotorSpeed <-> 1st RxPDO Mapping/Max motor speed
//     PlcTask Outputs/.P1_100_UG05.PDOS.PlcToDrv.maxTorque <-> 1st RxPDO Mapping/Max torque
//     PlcTask Outputs/.P1_100_UG05.PDOS.PlcToDrv.modesOfOperation <-> 1st RxPDO Mapping/Modes of operation
//     PlcTask Outputs/.P1_100_UG05.PDOS.PlcToDrv.vlTargetVelocity <-> 1st RxPDO Mapping/vl target velocity
//   Plc_Prog/Plc_Prog Instance <-> ETH/+P3=300-UG1 - WirePit Pump
//     PlcTask Inputs/.P1_100_UG02.PDOS.DrvToPLC.errorCode <-> 1st TxPDO Mapping/Error code
//     PlcTask Inputs/.P1_100_UG02.PDOS.DrvToPLC.modesOfOperationDisplay <-> 1st TxPDO Mapping/Mode Of Operation Display
//     PlcTask Inputs/.P1_100_UG02.PDOS.DrvToPLC.positionActualValue <-> 1st TxPDO Mapping/Position actual value
//     PlcTask Inputs/.P1_100_UG02.PDOS.DrvToPLC.statusWord <-> 1st TxPDO Mapping/Status Word
//     PlcTask Inputs/.P1_100_UG02.PDOS.DrvToPLC.torqueActualValue <-> 1st TxPDO Mapping/Torque actual value
//     PlcTask Inputs/.P1_100_UG02.PDOS.DrvToPLC.velocityActualValue <-> 1st TxPDO Mapping/Velocity actual value
//     PlcTask Outputs/.P1_100_UG02.PDOS.PlcToDrv.controlWord <-> 1st RxPDO Mapping/Control Word
//     PlcTask Outputs/.P1_100_UG02.PDOS.PlcToDrv.maxMotorSpeed <-> 1st RxPDO Mapping/Max motor speed
//     PlcTask Outputs/.P1_100_UG02.PDOS.PlcToDrv.maxTorque <-> 1st RxPDO Mapping/Max torque
//     PlcTask Outputs/.P1_100_UG02.PDOS.PlcToDrv.modesOfOperation <-> 1st RxPDO Mapping/Modes of operation
//     PlcTask Outputs/.P1_100_UG02.PDOS.PlcToDrv.vlTargetVelocity <-> 1st RxPDO Mapping/vl target velocity
//   Plc_Prog/Plc_Prog Instance <-> ETH/+P4=300-UG1 - Mix Pump
//     PlcTask Inputs/.P1_100_UG01.PDOS.DrvToPLC.errorCode <-> 1st TxPDO Mapping/Error code
//     PlcTask Inputs/.P1_100_UG01.PDOS.DrvToPLC.modesOfOperationDisplay <-> 1st TxPDO Mapping/Mode Of Operation Display
//     PlcTask Inputs/.P1_100_UG01.PDOS.DrvToPLC.positionActualValue <-> 1st TxPDO Mapping/Position actual value
//     PlcTask Inputs/.P1_100_UG01.PDOS.DrvToPLC.statusWord <-> 1st TxPDO Mapping/Status Word
//     PlcTask Inputs/.P1_100_UG01.PDOS.DrvToPLC.torqueActualValue <-> 1st TxPDO Mapping/Torque actual value
//     PlcTask Inputs/.P1_100_UG01.PDOS.DrvToPLC.velocityActualValue <-> 1st TxPDO Mapping/Velocity actual value
//     PlcTask Outputs/.P1_100_UG01.PDOS.PlcToDrv.controlWord <-> 1st RxPDO Mapping/Control Word
//     PlcTask Outputs/.P1_100_UG01.PDOS.PlcToDrv.maxMotorSpeed <-> 1st RxPDO Mapping/Max motor speed
//     PlcTask Outputs/.P1_100_UG01.PDOS.PlcToDrv.maxTorque <-> 1st RxPDO Mapping/Max torque
//     PlcTask Outputs/.P1_100_UG01.PDOS.PlcToDrv.modesOfOperation <-> 1st RxPDO Mapping/Modes of operation
//     PlcTask Outputs/.P1_100_UG01.PDOS.PlcToDrv.vlTargetVelocity <-> 1st RxPDO Mapping/vl target velocity
//   Plc_Prog/Plc_Prog Instance <-> ETH/+P5=050-BC1 - PLC Cabinet/+P5=050-DI1 (EL1809)
//     PlcTask Inputs/.P1_050_DI1.PDOS.digitalInput_01 <-> Channel 1/Input
//     PlcTask Inputs/.P1_050_DI1.PDOS.digitalInput_02 <-> Channel 2/Input
//     PlcTask Inputs/.P1_050_DI1.PDOS.digitalInput_03 <-> Channel 3/Input
//     PlcTask Inputs/.P1_050_DI1.PDOS.digitalInput_04 <-> Channel 4/Input
//     PlcTask Inputs/.P1_050_DI1.PDOS.digitalInput_05 <-> Channel 5/Input
//     PlcTask Inputs/.P1_050_DI1.PDOS.digitalInput_06 <-> Channel 6/Input
//     PlcTask Inputs/.P1_050_DI1.PDOS.digitalInput_07 <-> Channel 7/Input
//     PlcTask Inputs/.P1_050_DI1.PDOS.digitalInput_08 <-> Channel 8/Input
//     PlcTask Inputs/.P1_050_DI1.PDOS.digitalInput_09 <-> Channel 9/Input
//     PlcTask Inputs/.P1_050_DI1.PDOS.digitalInput_10 <-> Channel 10/Input
//     PlcTask Inputs/.P1_050_DI1.PDOS.digitalInput_11 <-> Channel 11/Input
//     PlcTask Inputs/.P1_050_DI1.PDOS.digitalInput_12 <-> Channel 12/Input
//     PlcTask Inputs/.P1_050_DI1.PDOS.digitalInput_13 <-> Channel 13/Input
//     PlcTask Inputs/.P1_050_DI1.PDOS.digitalInput_14 <-> Channel 14/Input
//     PlcTask Inputs/.P1_050_DI1.PDOS.digitalInput_15 <-> Channel 15/Input
//     PlcTask Inputs/.P1_050_DI1.PDOS.digitalInput_16 <-> Channel 16/Input
//   Plc_Prog/Plc_Prog Instance <-> ETH/+P5=050-BC1 - PLC Cabinet/+P5=050-DI2 (EL1809)
//     PlcTask Inputs/.P1_050_DI2.PDOS.digitalInput_01 <-> Channel 1/Input
//     PlcTask Inputs/.P1_050_DI2.PDOS.digitalInput_02 <-> Channel 2/Input
//     PlcTask Inputs/.P1_050_DI2.PDOS.digitalInput_03 <-> Channel 3/Input
//     PlcTask Inputs/.P1_050_DI2.PDOS.digitalInput_04 <-> Channel 4/Input
//     PlcTask Inputs/.P1_050_DI2.PDOS.digitalInput_05 <-> Channel 5/Input
//     PlcTask Inputs/.P1_050_DI2.PDOS.digitalInput_06 <-> Channel 6/Input
//     PlcTask Inputs/.P1_050_DI2.PDOS.digitalInput_07 <-> Channel 7/Input
//     PlcTask Inputs/.P1_050_DI2.PDOS.digitalInput_08 <-> Channel 8/Input
//     PlcTask Inputs/.P1_050_DI2.PDOS.digitalInput_09 <-> Channel 9/Input
//     PlcTask Inputs/.P1_050_DI2.PDOS.digitalInput_10 <-> Channel 10/Input
//     PlcTask Inputs/.P1_050_DI2.PDOS.digitalInput_13 <-> Channel 13/Input
//     PlcTask Inputs/.P1_050_DI2.PDOS.digitalInput_14 <-> Channel 14/Input
//     PlcTask Inputs/.P1_050_DI2.PDOS.digitalInput_15 <-> Channel 15/Input
//     PlcTask Inputs/.P1_050_DI2.PDOS.digitalInput_16 <-> Channel 16/Input
//     PlcTask Inputs/.P1_050_DI2.PDOS.digitalInput_11 <-> Channel 11/.P1_050_DI2.PDOS.digitalInput_11
//     PlcTask Inputs/.P1_050_DI2.PDOS.digitalInput_12 <-> Channel 12/.P1_050_DI2.PDOS.digitalInput_12
//   Plc_Prog/Plc_Prog Instance <-> ETH/+P5=050-BC1 - PLC Cabinet/+P5=050-DI3 (EL1809)
//     PlcTask Inputs/.P1_050_DI3.PDOS.digitalInput_01 <-> Channel 1/Input
//     PlcTask Inputs/.P1_050_DI3.PDOS.digitalInput_02 <-> Channel 2/Input
//     PlcTask Inputs/.P1_050_DI3.PDOS.digitalInput_03 <-> Channel 3/Input
//     PlcTask Inputs/.P1_050_DI3.PDOS.digitalInput_04 <-> Channel 4/Input
//     PlcTask Inputs/.P1_050_DI3.PDOS.digitalInput_05 <-> Channel 5/Input
//     PlcTask Inputs/.P1_050_DI3.PDOS.digitalInput_06 <-> Channel 6/Input
//     PlcTask Inputs/.P1_050_DI3.PDOS.digitalInput_07 <-> Channel 7/Input
//     PlcTask Inputs/.P1_050_DI3.PDOS.digitalInput_08 <-> Channel 8/Input
//     PlcTask Inputs/.P1_050_DI3.PDOS.digitalInput_09 <-> Channel 9/Input
//     PlcTask Inputs/.P1_050_DI3.PDOS.digitalInput_10 <-> Channel 10/Input
//     PlcTask Inputs/.P1_050_DI3.PDOS.digitalInput_11 <-> Channel 11/Input
//     PlcTask Inputs/.P1_050_DI3.PDOS.digitalInput_12 <-> Channel 12/Input
//     PlcTask Inputs/.P1_050_DI3.PDOS.digitalInput_13 <-> Channel 13/Input
//     PlcTask Inputs/.P1_050_DI3.PDOS.digitalInput_14 <-> Channel 14/Input
//     PlcTask Inputs/.P1_050_DI3.PDOS.digitalInput_15 <-> Channel 15/Input
//     PlcTask Inputs/.P1_050_DI3.PDOS.digitalInput_16 <-> Channel 16/Input
//   Plc_Prog/Plc_Prog Instance <-> ETH/+P5=050-BC1 - PLC Cabinet/+P5=050-DO1 (EL2809)
//     PlcTask Outputs/.P1_050_DO1.PDOS.PlcToHw.digitalOutput_01 <-> Channel 1/Output
//     PlcTask Outputs/.P1_050_DO1.PDOS.PlcToHw.digitalOutput_02 <-> Channel 2/Output
//     PlcTask Outputs/.P1_050_DO1.PDOS.PlcToHw.digitalOutput_03 <-> Channel 3/Output
//     PlcTask Outputs/.P1_050_DO1.PDOS.PlcToHw.digitalOutput_04 <-> Channel 4/Output
//     PlcTask Outputs/.P1_050_DO1.PDOS.PlcToHw.digitalOutput_05 <-> Channel 5/Output
//     PlcTask Outputs/.P1_050_DO1.PDOS.PlcToHw.digitalOutput_06 <-> Channel 6/Output
//     PlcTask Outputs/.P1_050_DO1.PDOS.PlcToHw.digitalOutput_07 <-> Channel 7/Output
//     PlcTask Outputs/.P1_050_DO1.PDOS.PlcToHw.digitalOutput_08 <-> Channel 8/Output
//     PlcTask Outputs/.P1_050_DO1.PDOS.PlcToHw.digitalOutput_09 <-> Channel 9/Output
//     PlcTask Outputs/.P1_050_DO1.PDOS.PlcToHw.digitalOutput_10 <-> Channel 10/Output
//     PlcTask Outputs/.P1_050_DO1.PDOS.PlcToHw.digitalOutput_11 <-> Channel 11/Output
//     PlcTask Outputs/.P1_050_DO1.PDOS.PlcToHw.digitalOutput_12 <-> Channel 12/Output
//     PlcTask Outputs/.P1_050_DO1.PDOS.PlcToHw.digitalOutput_13 <-> Channel 13/Output
//     PlcTask Outputs/.P1_050_DO1.PDOS.PlcToHw.digitalOutput_14 <-> Channel 14/Output
//     PlcTask Outputs/.P1_050_DO1.PDOS.PlcToHw.digitalOutput_15 <-> Channel 15/Output
//     PlcTask Outputs/.P1_050_DO1.PDOS.PlcToHw.digitalOutput_16 <-> Channel 16/Output
//   Plc_Prog/Plc_Prog Instance <-> ETH/+P5=050-BC1 - PLC Cabinet/+P5=050-DO2 (EL2809)
//     PlcTask Outputs/.P1_050_DO2.PDOS.PlcToHw.digitalOutput_01 <-> Channel 1/Output
//     PlcTask Outputs/.P1_050_DO2.PDOS.PlcToHw.digitalOutput_02 <-> Channel 2/Output
//     PlcTask Outputs/.P1_050_DO2.PDOS.PlcToHw.digitalOutput_03 <-> Channel 3/Output
//     PlcTask Outputs/.P1_050_DO2.PDOS.PlcToHw.digitalOutput_04 <-> Channel 4/Output
//     PlcTask Outputs/.P1_050_DO2.PDOS.PlcToHw.digitalOutput_05 <-> Channel 5/Output
//     PlcTask Outputs/.P1_050_DO2.PDOS.PlcToHw.digitalOutput_06 <-> Channel 6/Output
//     PlcTask Outputs/.P1_050_DO2.PDOS.PlcToHw.digitalOutput_07 <-> Channel 7/Output
//     PlcTask Outputs/.P1_050_DO2.PDOS.PlcToHw.digitalOutput_08 <-> Channel 8/Output
//     PlcTask Outputs/.P1_050_DO2.PDOS.PlcToHw.digitalOutput_09 <-> Channel 9/Output
//     PlcTask Outputs/.P1_050_DO2.PDOS.PlcToHw.digitalOutput_10 <-> Channel 10/Output
//     PlcTask Outputs/.P1_050_DO2.PDOS.PlcToHw.digitalOutput_11 <-> Channel 11/Output
//     PlcTask Outputs/.P1_050_DO2.PDOS.PlcToHw.digitalOutput_12 <-> Channel 12/Output
//     PlcTask Outputs/.P1_050_DO2.PDOS.PlcToHw.digitalOutput_13 <-> Channel 13/Output
//     PlcTask Outputs/.P1_050_DO2.PDOS.PlcToHw.digitalOutput_14 <-> Channel 14/Output
//     PlcTask Outputs/.P1_050_DO2.PDOS.PlcToHw.digitalOutput_15 <-> Channel 15/Output
//     PlcTask Outputs/.P1_050_DO2.PDOS.PlcToHw.digitalOutput_16 <-> Channel 16/Output
//   Plc_Prog/Plc_Prog Instance <-> ETH/+P5=050-BC1 - PLC Cabinet/+P5=050-DO3 (EL2809)
//     PlcTask Outputs/.P1_050_DO3.PDOS.PlcToHw.digitalOutput_01 <-> Channel 1/Output
//     PlcTask Outputs/.P1_050_DO3.PDOS.PlcToHw.digitalOutput_02 <-> Channel 2/Output
//     PlcTask Outputs/.P1_050_DO3.PDOS.PlcToHw.digitalOutput_03 <-> Channel 3/Output
//     PlcTask Outputs/.P1_050_DO3.PDOS.PlcToHw.digitalOutput_04 <-> Channel 4/Output
//     PlcTask Outputs/.P1_050_DO3.PDOS.PlcToHw.digitalOutput_05 <-> Channel 5/Output
//     PlcTask Outputs/.P1_050_DO3.PDOS.PlcToHw.digitalOutput_06 <-> Channel 6/Output
//     PlcTask Outputs/.P1_050_DO3.PDOS.PlcToHw.digitalOutput_07 <-> Channel 7/Output
//     PlcTask Outputs/.P1_050_DO3.PDOS.PlcToHw.digitalOutput_08 <-> Channel 8/Output
//     PlcTask Outputs/.P1_050_DO3.PDOS.PlcToHw.digitalOutput_09 <-> Channel 9/Output
//     PlcTask Outputs/.P1_050_DO3.PDOS.PlcToHw.digitalOutput_10 <-> Channel 10/Output
//     PlcTask Outputs/.P1_050_DO3.PDOS.PlcToHw.digitalOutput_11 <-> Channel 11/Output
//     PlcTask Outputs/.P1_050_DO3.PDOS.PlcToHw.digitalOutput_12 <-> Channel 12/Output
//     PlcTask Outputs/.P1_050_DO3.PDOS.PlcToHw.digitalOutput_13 <-> Channel 13/Output
//     PlcTask Outputs/.P1_050_DO3.PDOS.PlcToHw.digitalOutput_14 <-> Channel 14/Output
//     PlcTask Outputs/.P1_050_DO3.PDOS.PlcToHw.digitalOutput_15 <-> Channel 15/Output
//     PlcTask Outputs/.P1_050_DO3.PDOS.PlcToHw.digitalOutput_16 <-> Channel 16/Output
//   Plc_Prog/Plc_Prog Instance <-> ETH/+P5=050-BC1 - PLC Cabinet/+P5=050-SP1 (EL6910)
//     PlcTask Inputs/.P1_050_SP1.PDOS.HwToPLC.EStop1Diag <-> Function Block Info Data/TwinSafeGroup1.Network1.FBEstop1 Info Data/Diag
//     PlcTask Inputs/.P1_050_SP1.PDOS.HwToPLC.EStop2Diag <-> Function Block Info Data/TwinSafeGroup1.Network1.FBEstop2 Info Data/Diag
//     PlcTask Inputs/.P1_050_SP1.PDOS.HwToPLC.EStop3Diag <-> Function Block Info Data/TwinSafeGroup1.Network1.FBEstop3 Info Data/Diag
//     PlcTask Inputs/.P1_050_SP1.PDOS.HwToPLC.EStop1State <-> Function Block Info Data/TwinSafeGroup1.Network1.FBEstop1 Info Data/State
//     PlcTask Inputs/.P1_050_SP1.PDOS.HwToPLC.EStop2State <-> Function Block Info Data/TwinSafeGroup1.Network1.FBEstop2 Info Data/State
//     PlcTask Inputs/.P1_050_SP1.PDOS.HwToPLC.EStop3State <-> Function Block Info Data/TwinSafeGroup1.Network1.FBEstop3 Info Data/State
//     PlcTask Outputs/.P1_050_SP1.PDOS.PlcToHw.ErrorAcknowledgement <-> StandardOutputs/TwinSafeGroup1.ErrorAcknowledgement_1
//     PlcTask Outputs/.P1_050_SP1.PDOS.PlcToHw.Run <-> StandardOutputs/TwinSafeGroup1.Run_2
//     PlcTask Outputs/.P1_050_SP1.PDOS.PlcToHw.safetyReset <-> StandardOutputs/TwinSafeGroup1.SafetyReset_6
//   Plc_Prog/Plc_Prog Instance <-> ETH/+P5=050-BC2 - PLC Cabinet/+P5=050-AI (EL3052)
//     PlcTask Inputs/.P1_050_AI1.PDOS.HwToPLC.Channel1/Status/Error <-> AI Standard Channel 1/Status/TxPDO Toggle
//     PlcTask Inputs/.P1_050_AI1.PDOS.HwToPLC.Channel1/Status/Limit1 <-> AI Standard Channel 1/Status/Error
//     PlcTask Inputs/.P1_050_AI1.PDOS.HwToPLC.Channel1/Status/Limit2 <-> AI Standard Channel 1/Status/TxPDO State
//     PlcTask Inputs/.P1_050_AI1.PDOS.HwToPLC.Channel1/Status/Overrange <-> AI Standard Channel 1/Status/Overrange
//     PlcTask Inputs/.P1_050_AI1.PDOS.HwToPLC.Channel2/Status/Overrange <-> AI Standard Channel 2/Status/Overrange
//     PlcTask Inputs/.P1_050_AI1.PDOS.HwToPLC.Channel1/Status/Underrange <-> AI Standard Channel 1/Status/Underrange
//     PlcTask Inputs/.P1_050_AI1.PDOS.HwToPLC.Channel2/Status/Underrange <-> AI Standard Channel 2/Status/Underrange
//     PlcTask Inputs/.P1_050_AI1.PDOS.HwToPLC.Channel1/Value <-> AI Standard Channel 1/Value
//     PlcTask Inputs/.P1_050_AI1.PDOS.HwToPLC.Channel2/Value <-> AI Standard Channel 2/Value
//     PlcTask Inputs/.P1_050_AI1.PDOS.HwToPLC.Channel2/Status/Error <-> AI Standard Channel 2/Status/Error
//     PlcTask Inputs/.P1_050_AI1.PDOS.HwToPLC.Channel2/Status/TxPDOState <-> AI Standard Channel 2/Status/TxPDO State
//     PlcTask Inputs/.P1_050_AI1.PDOS.HwToPLC.Channel2/Status/TxPDOToggle <-> AI Standard Channel 2/Status/TxPDO Toggle
//   Plc_Prog/Plc_Prog Instance <-> ETH/+P5=050-BC2 - PLC Cabinet/+P5=050-AI2 (EL3152)
//     PlcTask Inputs/.P1_050_AI2.PDOS.HwToPLC.Channel1/Status/Error <-> AI Standard Channel 1/Status/Error
//     PlcTask Inputs/.P1_050_AI2.PDOS.HwToPLC.Channel2/Status/Error <-> AI Standard Channel 2/Status/Error
//     PlcTask Inputs/.P1_050_AI2.PDOS.HwToPLC.Channel1/Status/Overrange <-> AI Standard Channel 1/Status/Overrange
//     PlcTask Inputs/.P1_050_AI2.PDOS.HwToPLC.Channel2/Status/Overrange <-> AI Standard Channel 2/Status/Overrange
//     PlcTask Inputs/.P1_050_AI2.PDOS.HwToPLC.Channel1/Status/TxPDOState <-> AI Standard Channel 1/Status/TxPDO State
//     PlcTask Inputs/.P1_050_AI2.PDOS.HwToPLC.Channel2/Status/TxPDOState <-> AI Standard Channel 2/Status/TxPDO State
//     PlcTask Inputs/.P1_050_AI2.PDOS.HwToPLC.Channel1/Status/TxPDOToggle <-> AI Standard Channel 1/Status/TxPDO Toggle
//     PlcTask Inputs/.P1_050_AI2.PDOS.HwToPLC.Channel2/Status/TxPDOToggle <-> AI Standard Channel 2/Status/TxPDO Toggle
//     PlcTask Inputs/.P1_050_AI2.PDOS.HwToPLC.Channel1/Status/Underrange <-> AI Standard Channel 1/Status/Underrange
//     PlcTask Inputs/.P1_050_AI2.PDOS.HwToPLC.Channel2/Status/Underrange <-> AI Standard Channel 2/Status/Underrange
//     PlcTask Inputs/.P1_050_AI2.PDOS.HwToPLC.Channel1/Value <-> AI Standard Channel 1/Value
//     PlcTask Inputs/.P1_050_AI2.PDOS.HwToPLC.Channel2/Value <-> AI Standard Channel 2/Value
//   Plc_Prog/Plc_Prog Instance <-> ETH/+P5=050-BC2 - PLC Cabinet/+P5=050-AI3 (EL3052)
//     PlcTask Inputs/.P1_050_AI3.PDOS.HwToPLC.Channel1/Status/Error <-> AI Standard Channel 1/Status/Error
//     PlcTask Inputs/.P1_050_AI3.PDOS.HwToPLC.Channel2/Status/Error <-> AI Standard Channel 2/Status/Error
//     PlcTask Inputs/.P1_050_AI3.PDOS.HwToPLC.Channel1/Status/Overrange <-> AI Standard Channel 1/Status/Overrange
//     PlcTask Inputs/.P1_050_AI3.PDOS.HwToPLC.Channel2/Status/Overrange <-> AI Standard Channel 2/Status/Overrange
//     PlcTask Inputs/.P1_050_AI3.PDOS.HwToPLC.Channel1/Status/TxPDOState <-> AI Standard Channel 1/Status/TxPDO State
//     PlcTask Inputs/.P1_050_AI3.PDOS.HwToPLC.Channel2/Status/TxPDOState <-> AI Standard Channel 2/Status/TxPDO State
//     PlcTask Inputs/.P1_050_AI3.PDOS.HwToPLC.Channel1/Status/TxPDOToggle <-> AI Standard Channel 1/Status/TxPDO Toggle
//     PlcTask Inputs/.P1_050_AI3.PDOS.HwToPLC.Channel2/Status/TxPDOToggle <-> AI Standard Channel 2/Status/TxPDO Toggle
//     PlcTask Inputs/.P1_050_AI3.PDOS.HwToPLC.Channel1/Status/Underrange <-> AI Standard Channel 1/Status/Underrange
//     PlcTask Inputs/.P1_050_AI3.PDOS.HwToPLC.Channel2/Status/Underrange <-> AI Standard Channel 2/Status/Underrange
//     PlcTask Inputs/.P1_050_AI3.PDOS.HwToPLC.Channel1/Value <-> AI Standard Channel 1/Value
//     PlcTask Inputs/.P1_050_AI3.PDOS.HwToPLC.Channel2/Value <-> AI Standard Channel 2/Value
//   Plc_Prog/Plc_Prog Instance <-> ETH/+P5=050-BC2 - PLC Cabinet/+P5=050-AI4 (EL3052)
//     PlcTask Inputs/.P1_050_AI4.PDOS.HwToPLC.Channel1/Status/Error <-> AI Standard Channel 1/Status/Error
//     PlcTask Inputs/.P1_050_AI4.PDOS.HwToPLC.Channel2/Status/Error <-> AI Standard Channel 2/Status/Error
//     PlcTask Inputs/.P1_050_AI4.PDOS.HwToPLC.Channel1/Status/Overrange <-> AI Standard Channel 1/Status/Overrange
//     PlcTask Inputs/.P1_050_AI4.PDOS.HwToPLC.Channel2/Status/Overrange <-> AI Standard Channel 2/Status/Overrange
//     PlcTask Inputs/.P1_050_AI4.PDOS.HwToPLC.Channel1/Status/TxPDOState <-> AI Standard Channel 1/Status/TxPDO State
//     PlcTask Inputs/.P1_050_AI4.PDOS.HwToPLC.Channel2/Status/TxPDOState <-> AI Standard Channel 2/Status/TxPDO State
//     PlcTask Inputs/.P1_050_AI4.PDOS.HwToPLC.Channel1/Status/TxPDOToggle <-> AI Standard Channel 1/Status/TxPDO Toggle
//     PlcTask Inputs/.P1_050_AI4.PDOS.HwToPLC.Channel2/Status/TxPDOToggle <-> AI Standard Channel 2/Status/TxPDO Toggle
//     PlcTask Inputs/.P1_050_AI4.PDOS.HwToPLC.Channel1/Status/Underrange <-> AI Standard Channel 1/Status/Underrange
//     PlcTask Inputs/.P1_050_AI4.PDOS.HwToPLC.Channel2/Status/Underrange <-> AI Standard Channel 2/Status/Underrange
//     PlcTask Inputs/.P1_050_AI4.PDOS.HwToPLC.Channel1/Value <-> AI Standard Channel 1/Value
//     PlcTask Inputs/.P1_050_AI4.PDOS.HwToPLC.Channel2/Value <-> AI Standard Channel 2/Value
//   Plc_Prog/Plc_Prog Instance <-> ETH/+P9=050-BC1 - Vaccum PLC Cabinet/+P9=050-AI1 (EL3054)
//     PlcTask Inputs/.P9_050_AI1.PDOS.HwToPLC.Channel1/Status/Error <-> AI Standard Channel 1/Status/Error
//     PlcTask Inputs/.P9_050_AI1.PDOS.HwToPLC.Channel2/Status/Error <-> AI Standard Channel 2/Status/Error
//     PlcTask Inputs/.P9_050_AI1.PDOS.HwToPLC.Channel1/Status/Overrange <-> AI Standard Channel 1/Status/Overrange
//     PlcTask Inputs/.P9_050_AI1.PDOS.HwToPLC.Channel2/Status/Overrange <-> AI Standard Channel 2/Status/Overrange
//     PlcTask Inputs/.P9_050_AI1.PDOS.HwToPLC.Channel1/Status/TxPDOState <-> AI Standard Channel 1/Status/TxPDO State
//     PlcTask Inputs/.P9_050_AI1.PDOS.HwToPLC.Channel2/Status/TxPDOState <-> AI Standard Channel 2/Status/TxPDO State
//     PlcTask Inputs/.P9_050_AI1.PDOS.HwToPLC.Channel1/Status/TxPDOToggle <-> AI Standard Channel 1/Status/TxPDO Toggle
//     PlcTask Inputs/.P9_050_AI1.PDOS.HwToPLC.Channel2/Status/TxPDOToggle <-> AI Standard Channel 2/Status/TxPDO Toggle
//     PlcTask Inputs/.P9_050_AI1.PDOS.HwToPLC.Channel1/Status/Underrange <-> AI Standard Channel 1/Status/Underrange
//     PlcTask Inputs/.P9_050_AI1.PDOS.HwToPLC.Channel2/Status/Underrange <-> AI Standard Channel 2/Status/Underrange
//     PlcTask Inputs/.P9_050_AI1.PDOS.HwToPLC.Channel1/Value <-> AI Standard Channel 1/Value
//     PlcTask Inputs/.P9_050_AI1.PDOS.HwToPLC.Channel2/Value <-> AI Standard Channel 2/Value
//   Plc_Prog/Plc_Prog Instance <-> ETH/+P9=050-BC1 - Vaccum PLC Cabinet/+P9=050-DI1 (EL1809)
//     PlcTask Inputs/.P9_050_DI1.PDOS.digitalInput_01 <-> Channel 1/Input
//     PlcTask Inputs/.P9_050_DI1.PDOS.digitalInput_02 <-> Channel 2/Input
//     PlcTask Inputs/.P9_050_DI1.PDOS.digitalInput_03 <-> Channel 3/Input
//     PlcTask Inputs/.P9_050_DI1.PDOS.digitalInput_04 <-> Channel 4/Input
//     PlcTask Inputs/.P9_050_DI1.PDOS.digitalInput_05 <-> Channel 5/Input
//     PlcTask Inputs/.P9_050_DI1.PDOS.digitalInput_06 <-> Channel 6/Input
//     PlcTask Inputs/.P9_050_DI1.PDOS.digitalInput_07 <-> Channel 7/Input
//     PlcTask Inputs/.P9_050_DI1.PDOS.digitalInput_08 <-> Channel 8/Input
//     PlcTask Inputs/.P9_050_DI1.PDOS.digitalInput_09 <-> Channel 9/Input
//     PlcTask Inputs/.P9_050_DI1.PDOS.digitalInput_10 <-> Channel 10/Input
//     PlcTask Inputs/.P9_050_DI1.PDOS.digitalInput_11 <-> Channel 11/Input
//     PlcTask Inputs/.P9_050_DI1.PDOS.digitalInput_12 <-> Channel 12/Input
//     PlcTask Inputs/.P9_050_DI1.PDOS.digitalInput_13 <-> Channel 13/Input
//     PlcTask Inputs/.P9_050_DI1.PDOS.digitalInput_14 <-> Channel 14/Input
//     PlcTask Inputs/.P9_050_DI1.PDOS.digitalInput_15 <-> Channel 15/Input
//     PlcTask Inputs/.P9_050_DI1.PDOS.digitalInput_16 <-> Channel 16/Input
//   Plc_Prog/Plc_Prog Instance <-> ETH/+P9=050-BC1 - Vaccum PLC Cabinet/+P9=050-DI2 (EL1809)
//     PlcTask Inputs/.P9_050_DI2.PDOS.digitalInput_01 <-> Channel 1/Input
//     PlcTask Inputs/.P9_050_DI2.PDOS.digitalInput_02 <-> Channel 2/Input
//     PlcTask Inputs/.P9_050_DI2.PDOS.digitalInput_03 <-> Channel 3/Input
//     PlcTask Inputs/.P9_050_DI2.PDOS.digitalInput_04 <-> Channel 4/Input
//     PlcTask Inputs/.P9_050_DI2.PDOS.digitalInput_05 <-> Channel 5/Input
//     PlcTask Inputs/.P9_050_DI2.PDOS.digitalInput_06 <-> Channel 6/Input
//     PlcTask Inputs/.P9_050_DI2.PDOS.digitalInput_07 <-> Channel 7/Input
//     PlcTask Inputs/.P9_050_DI2.PDOS.digitalInput_08 <-> Channel 8/Input
//     PlcTask Inputs/.P9_050_DI2.PDOS.digitalInput_09 <-> Channel 9/Input
//     PlcTask Inputs/.P9_050_DI2.PDOS.digitalInput_10 <-> Channel 10/Input
//     PlcTask Inputs/.P9_050_DI2.PDOS.digitalInput_11 <-> Channel 11/Input
//     PlcTask Inputs/.P9_050_DI2.PDOS.digitalInput_12 <-> Channel 12/Input
//     PlcTask Inputs/.P9_050_DI2.PDOS.digitalInput_13 <-> Channel 13/Input
//     PlcTask Inputs/.P9_050_DI2.PDOS.digitalInput_14 <-> Channel 14/Input
//     PlcTask Inputs/.P9_050_DI2.PDOS.digitalInput_15 <-> Channel 15/Input
//     PlcTask Inputs/.P9_050_DI2.PDOS.digitalInput_16 <-> Channel 16/Input
//   Plc_Prog/Plc_Prog Instance <-> ETH/+P9=050-BC1 - Vaccum PLC Cabinet/+P9=050-DI3 (EL1809)
//     PlcTask Inputs/.P9_050_DI3.PDOS.digitalInput_01 <-> Channel 1/Input
//     PlcTask Inputs/.P9_050_DI3.PDOS.digitalInput_02 <-> Channel 2/Input
//     PlcTask Inputs/.P9_050_DI3.PDOS.digitalInput_03 <-> Channel 3/Input
//     PlcTask Inputs/.P9_050_DI3.PDOS.digitalInput_04 <-> Channel 4/Input
//     PlcTask Inputs/.P9_050_DI3.PDOS.digitalInput_05 <-> Channel 5/Input
//     PlcTask Inputs/.P9_050_DI3.PDOS.digitalInput_06 <-> Channel 6/Input
//     PlcTask Inputs/.P9_050_DI3.PDOS.digitalInput_07 <-> Channel 7/Input
//     PlcTask Inputs/.P9_050_DI3.PDOS.digitalInput_08 <-> Channel 8/Input
//     PlcTask Inputs/.P9_050_DI3.PDOS.digitalInput_09 <-> Channel 9/Input
//     PlcTask Inputs/.P9_050_DI3.PDOS.digitalInput_10 <-> Channel 10/Input
//     PlcTask Inputs/.P9_050_DI3.PDOS.digitalInput_11 <-> Channel 11/Input
//     PlcTask Inputs/.P9_050_DI3.PDOS.digitalInput_12 <-> Channel 12/Input
//     PlcTask Inputs/.P9_050_DI3.PDOS.digitalInput_13 <-> Channel 13/Input
//     PlcTask Inputs/.P9_050_DI3.PDOS.digitalInput_14 <-> Channel 14/Input
//     PlcTask Inputs/.P9_050_DI3.PDOS.digitalInput_15 <-> Channel 15/Input
//     PlcTask Inputs/.P9_050_DI3.PDOS.digitalInput_16 <-> Channel 16/Input
//   Plc_Prog/Plc_Prog Instance <-> ETH/+P9=050-BC1 - Vaccum PLC Cabinet/+P9=050-DO1 (EL2809)
//     PlcTask Outputs/.P9_050_DO1.PDOS.PlcToHw.digitalOutput_01 <-> Channel 1/Output
//     PlcTask Outputs/.P9_050_DO1.PDOS.PlcToHw.digitalOutput_02 <-> Channel 2/Output
//     PlcTask Outputs/.P9_050_DO1.PDOS.PlcToHw.digitalOutput_03 <-> Channel 3/Output
//     PlcTask Outputs/.P9_050_DO1.PDOS.PlcToHw.digitalOutput_04 <-> Channel 4/Output
//     PlcTask Outputs/.P9_050_DO1.PDOS.PlcToHw.digitalOutput_05 <-> Channel 5/Output
//     PlcTask Outputs/.P9_050_DO1.PDOS.PlcToHw.digitalOutput_06 <-> Channel 6/Output
//     PlcTask Outputs/.P9_050_DO1.PDOS.PlcToHw.digitalOutput_07 <-> Channel 7/Output
//     PlcTask Outputs/.P9_050_DO1.PDOS.PlcToHw.digitalOutput_08 <-> Channel 8/Output
//     PlcTask Outputs/.P9_050_DO1.PDOS.PlcToHw.digitalOutput_09 <-> Channel 9/Output
//     PlcTask Outputs/.P9_050_DO1.PDOS.PlcToHw.digitalOutput_10 <-> Channel 10/Output
//     PlcTask Outputs/.P9_050_DO1.PDOS.PlcToHw.digitalOutput_11 <-> Channel 11/Output
//     PlcTask Outputs/.P9_050_DO1.PDOS.PlcToHw.digitalOutput_12 <-> Channel 12/Output
//     PlcTask Outputs/.P9_050_DO1.PDOS.PlcToHw.digitalOutput_13 <-> Channel 13/Output
//     PlcTask Outputs/.P9_050_DO1.PDOS.PlcToHw.digitalOutput_14 <-> Channel 14/Output
//     PlcTask Outputs/.P9_050_DO1.PDOS.PlcToHw.digitalOutput_15 <-> Channel 15/Output
//     PlcTask Outputs/.P9_050_DO1.PDOS.PlcToHw.digitalOutput_16 <-> Channel 16/Output
//   Plc_Prog/Plc_Prog Instance <-> ETH/+P9=050-BC1 - Vaccum PLC Cabinet/+P9=050-DO2 (EL2809)
//     PlcTask Outputs/.P9_050_DO2.PDOS.PlcToHw.digitalOutput_01 <-> Channel 1/Output
//     PlcTask Outputs/.P9_050_DO2.PDOS.PlcToHw.digitalOutput_02 <-> Channel 2/Output
//     PlcTask Outputs/.P9_050_DO2.PDOS.PlcToHw.digitalOutput_03 <-> Channel 3/Output
//     PlcTask Outputs/.P9_050_DO2.PDOS.PlcToHw.digitalOutput_04 <-> Channel 4/Output
//     PlcTask Outputs/.P9_050_DO2.PDOS.PlcToHw.digitalOutput_05 <-> Channel 5/Output
//     PlcTask Outputs/.P9_050_DO2.PDOS.PlcToHw.digitalOutput_06 <-> Channel 6/Output
//     PlcTask Outputs/.P9_050_DO2.PDOS.PlcToHw.digitalOutput_07 <-> Channel 7/Output
//     PlcTask Outputs/.P9_050_DO2.PDOS.PlcToHw.digitalOutput_08 <-> Channel 8/Output
//     PlcTask Outputs/.P9_050_DO2.PDOS.PlcToHw.digitalOutput_09 <-> Channel 9/Output
//     PlcTask Outputs/.P9_050_DO2.PDOS.PlcToHw.digitalOutput_10 <-> Channel 10/Output
//     PlcTask Outputs/.P9_050_DO2.PDOS.PlcToHw.digitalOutput_11 <-> Channel 11/Output
//     PlcTask Outputs/.P9_050_DO2.PDOS.PlcToHw.digitalOutput_12 <-> Channel 12/Output
//     PlcTask Outputs/.P9_050_DO2.PDOS.PlcToHw.digitalOutput_13 <-> Channel 13/Output
//     PlcTask Outputs/.P9_050_DO2.PDOS.PlcToHw.digitalOutput_14 <-> Channel 14/Output
//     PlcTask Outputs/.P9_050_DO2.PDOS.PlcToHw.digitalOutput_15 <-> Channel 15/Output
//     PlcTask Outputs/.P9_050_DO2.PDOS.PlcToHw.digitalOutput_16 <-> Channel 16/Output
//   Plc_Prog/Plc_Prog Instance <-> ETH/+P9=050-BC1 - Vaccum PLC Cabinet/+P9=050-DO3 (EL2809)
//     PlcTask Outputs/.P9_050_DO3.PDOS.PlcToHw.digitalOutput_01 <-> Channel 1/Output
//     PlcTask Outputs/.P9_050_DO3.PDOS.PlcToHw.digitalOutput_02 <-> Channel 2/Output
//     PlcTask Outputs/.P9_050_DO3.PDOS.PlcToHw.digitalOutput_06 <-> Channel 6/Output
//     PlcTask Outputs/.P9_050_DO3.PDOS.PlcToHw.digitalOutput_07 <-> Channel 7/Output
//     PlcTask Outputs/.P9_050_DO3.PDOS.PlcToHw.digitalOutput_08 <-> Channel 8/Output
//     PlcTask Outputs/.P9_050_DO3.PDOS.PlcToHw.digitalOutput_09 <-> Channel 9/Output
//     PlcTask Outputs/.P9_050_DO3.PDOS.PlcToHw.digitalOutput_10 <-> Channel 10/Output
//     PlcTask Outputs/.P9_050_DO3.PDOS.PlcToHw.digitalOutput_11 <-> Channel 11/Output
//     PlcTask Outputs/.P9_050_DO3.PDOS.PlcToHw.digitalOutput_12 <-> Channel 12/Output
//     PlcTask Outputs/.P9_050_DO3.PDOS.PlcToHw.digitalOutput_13 <-> Channel 13/Output
//     PlcTask Outputs/.P9_050_DO3.PDOS.PlcToHw.digitalOutput_14 <-> Channel 14/Output
//     PlcTask Outputs/.P9_050_DO3.PDOS.PlcToHw.digitalOutput_15 <-> Channel 15/Output
//     PlcTask Outputs/.P9_050_DO3.PDOS.PlcToHw.digitalOutput_16 <-> Channel 16/Output
//     PlcTask Outputs/.P9_050_DO3.PDOS.PlcToHw.digitalOutput_03 <-> Channel 3/Libera Safety Vacuo
//     PlcTask Outputs/.P9_050_DO3.PDOS.PlcToHw.digitalOutput_04 <-> Channel 4/Selagem do vacuo
//     PlcTask Outputs/.P9_050_DO3.PDOS.PlcToHw.digitalOutput_05 <-> Channel 5/Separador Baixo Vacuo
//   Plc_Prog/Plc_Prog Instance <-> ETH/+P9=050-BC1 - Vaccum PLC Cabinet/Term 101 (EL3052)
//     PlcTask Inputs/.P9_050_AI2.PDOS.HwToPLC.Channel1/Status/Overrange <-> AI Standard Channel 1/Status/Overrange
//     PlcTask Inputs/.P9_050_AI2.PDOS.HwToPLC.Channel1/Status/Underrange <-> AI Standard Channel 1/Status/Underrange
//     PlcTask Inputs/.P9_050_AI2.PDOS.HwToPLC.Channel1/Value <-> AI Standard Channel 1/Value
//     PlcTask Inputs/.P9_050_AI2.PDOS.HwToPLC.Channel2/Value <-> AI Standard Channel 2/Value
//     PlcTask Inputs/.P9_050_AI2.PDOS.HwToPLC.Channel2/Status/Overrange <-> AI Standard Channel 2/Status/Underrange
//   Plc_Prog/Plc_Prog Instance <-> ETH/+P9=050-BC1 - Vaccum PLC Cabinet/Term 102 (EL4004)
//     PlcTask Outputs/.P9_050_AQ1.PDOS.HwToPLC.Channel1 <-> AO Outputs Channel 1/Analog output
//     PlcTask Outputs/.P9_050_AQ1.PDOS.HwToPLC.Channel2 <-> AO Outputs Channel 2/Analog output
//     PlcTask Outputs/.P9_050_AQ1.PDOS.HwToPLC.Channel3 <-> AO Outputs Channel 3/Analog output
//     PlcTask Outputs/.P9_050_AQ1.PDOS.HwToPLC.Channel4 <-> AO Outputs Channel 4/Analog output

CONFIGURATION Plc_Prog
    RESOURCE PLC ON TwinCAT3
        TASK PlcTask(INTERVAL := T#5ms, PRIORITY := 20);
        PROGRAM MAIN WITH PlcTask : MAIN;
    END_RESOURCE
END_CONFIGURATION

// ---- Function Blocks/DELTA - MS300/C2000_ANALOG_INPUTS.TcDUT
TYPE C2000_ANALOG_INPUTS :
STRUCT
	
	AVI : REAL;
	ACI : REAL;

END_STRUCT
END_TYPE

// ---- Function Blocks/DELTA - MS300/C2000_ANALOG_OUTPUTS.TcDUT
TYPE C2000_ANALOG_OUTPUTS :
STRUCT
	
	AFM : REAL;

END_STRUCT
END_TYPE

// ---- Function Blocks/DELTA - MS300/C2000_CONTROLWORD.TcDUT
TYPE C2000_CONTROLWORD :
STRUCT
	
    enableDrive     : BOOL;   // request to run (Enable Operation)
    stopRequest     : BOOL;   // keep voltage on but do not enable operation
    quickStop       : BOOL;   // immediate controlled stop (bit2 = 0)
    halt            : BOOL;   // CiA-402 halt (bit8 = 1)
    faultResetCmd   : BOOL;   // pulse fault reset
		
END_STRUCT
END_TYPE

// ---- Function Blocks/DELTA - MS300/C2000_DIGITAL_OUTPUTS.TcDUT
TYPE C2000_DIGITAL_OUTPUTS :
STRUCT
		
	RLY					: BOOL; (*Drive relay output - Terminal RLY*)
	MO1					: BOOL; (*Drive digital output - Terminal MO2*)
	MO2					: BOOL; (*Drive digital output - Terminal MO3*)
		
END_STRUCT
END_TYPE

// ---- Function Blocks/DELTA - MS300/C2000_DRVTOPLC_PDOS.TcDUT
TYPE C2000_DRVTOPLC_PDOS :
	STRUCT	
		
		statusWord              AT %I* : UINT;   //Status word of the drive
		errorCode               AT %I*: UINT;   //Error code of the drive
		modesOfOperationDisplay AT %I*: SINT;   //Current mode of operation
		positionActualValue     AT %I*: DINT;   //Actual position feedback
		velocityActualValue     AT %I*: DINT;   //Actual velocity feedback
		torqueActualValue       AT %I*: INT;    //Actual torque feedback
		
	END_STRUCT
END_TYPE

// ---- Function Blocks/DELTA - MS300/C2000_PLCTODRV_PDOS.TcDUT
TYPE C2000_PLCTODRV_PDOS :
    STRUCT
		
		controlWord       AT %Q* : UINT;   // Control word to command the drive
		vlTargetVelocity  AT %Q*: INT;    // Target velocity [vl = velocity]
		modesOfOperation  AT %Q* : SINT;   // Mode of operation command
		maxTorque         AT %Q* : UINT;   // Maximum torque limit
		maxMotorSpeed     AT %Q* : UDINT;  // Maximum motor speed limit

    END_STRUCT
END_TYPE
(*


	digitalInput_11 AT %I* : BOOL;
	digitalInput_12 AT %I* : BOOL;
	digitalInput_13 AT %I* : BOOL;
	digitalInput_14 AT %I* : BOOL;
	digitalInput_15 AT %I* : BOOL;


*)

// ---- Function Blocks/DELTA - MS300/C2000_STATUSWORD.TcDUT
(*TYPE C2000_STATUSWORD :
    STRUCT
        notRunning      : BOOL; // Indicates if the drive is not running
        running         : BOOL; // Indicates if the drive is running
        jogging         : BOOL; // Indicates if the drive is in jogging mode
        runningForward  : BOOL; // Indicates if the drive is running forward
        runningReverse  : BOOL; // Indicates if the drive is running in reverse
        fault           : BOOL; // Indicates if there is a fault in the drive
    END_STRUCT
END_TYPE
*)
TYPE C2000_STATUSWORD :
STRUCT
    readyToSwitchOn     : BOOL; // Bit 0 - Drive is ready to switch on
    switchedOn          : BOOL; // Bit 1 - Drive is switched on
    operationEnabled    : BOOL; // Bit 2 - Operation enabled
    fault               : BOOL; // Bit 3 - Fault present
    voltageEnabled      : BOOL; // Bit 4 - DC bus / power voltage enabled
    quickStop           : BOOL; // Bit 5 - Quick stop active
    switchOnDisabled    : BOOL; // Bit 6 - Switch on disabled

    warning             : BOOL; // Bit 7 - Warning, servo remains on
    reserved1           : BOOL; // Bit 8 - Reserved
    remote              : BOOL; // Bit 9 - Drive in remote (fieldbus) mode
    targetReached       : BOOL; // Bit 10 - Target position reached
    internalLimitActive : BOOL; // Bit 11 - Software limit active
    operationModeSpec   : WORD; // Bit 12–13 - Operation mode specific (2 bits wide)
    externalLimitActive : BOOL; // Bit 14 - Hardware limit active
    reserved2           : BOOL; // Bit 15 - Reserved
END_STRUCT
END_TYPE

// ---- Function Blocks/IOs/Beckhoff/EL1809 - Digital Inputs/DataTypes/EL1809_HWTOPLC_PDOS.TcDUT
TYPE EL1809_HWTOPLC_PDOS :
	STRUCT
		
	
	digitalInput_01 AT %I* : BOOL;
	digitalInput_02 AT %I* : BOOL;
	digitalInput_03 AT %I* : BOOL;
	digitalInput_04 AT %I* : BOOL;
	digitalInput_05 AT %I* : BOOL;
	digitalInput_06 AT %I* : BOOL;
	digitalInput_07 AT %I* : BOOL;
	digitalInput_08 AT %I* : BOOL;
	digitalInput_09 AT %I* : BOOL;
	digitalInput_10 AT %I* : BOOL;
	digitalInput_11 AT %I* : BOOL;
	digitalInput_12 AT %I* : BOOL;
	digitalInput_13 AT %I* : BOOL;
	digitalInput_14 AT %I* : BOOL;
	digitalInput_15 AT %I* : BOOL;
	digitalInput_16 AT %I* : BOOL;


		
	END_STRUCT
END_TYPE

// ---- Function Blocks/IOs/Beckhoff/EL3052 - Ai 2 x 4-20MA - 12bit/DataTypes/EL3052_DEV_CONFIG.TcDUT
TYPE EL3052_DEV_CONFIG :
    STRUCT
   
        // Setpoint scaling
       	channel1InputLow        : REAL := 0.0;   // Minimum input value for setpoint		
        channel1InputHigh       : REAL := 30518.0; // Maximum input value for setpoint
        channel1OutputLow       : REAL := 0.0; // Minimum output value for setpoint
        channel1OutputHigh      : REAL := 100.0; // Maximum output value for setpoint
        // Setpoint scaling
       	channe12InputLow        : REAL := 0.0;   // Minimum input value for setpoint		
        channe12InputHigh       : REAL := 30518.0; // Maximum input value for setpoint
        channe12OutputLow       : REAL := 0.0; // Minimum output value for setpoint
        channe12OutputHigh      : REAL := 100.0; // Maximum output value for setpoint		

    END_STRUCT
END_TYPE

// ---- Function Blocks/IOs/Beckhoff/EL3052 - Ai 2 x 4-20MA - 12bit/DataTypes/EL3052_DEV_STATUS.TcDUT
TYPE EL3052_DEV_STATUS :
    STRUCT
      
		Underrange : BOOL;
		Overrange : BOOL;
		Limit1 : BOOL;
		Limit2 : BOOL;
		Error : BOOL;
		TxPDOState : BOOL;
		TxPDOToggle : BOOL;
	
    END_STRUCT
END_TYPE

// ---- Function Blocks/IOs/Beckhoff/EL3052 - Ai 2 x 4-20MA - 12bit/DataTypes/EL3052_HWTOPLC_PDOS.TcDUT
TYPE EL3052_HWTOPLC_PDOS :
	STRUCT
		
	
	Channel1 	AT %I* : EL3052_CHANNEL;
	Channel2 	AT %I* : EL3052_CHANNEL;



	END_STRUCT
END_TYPE

// ---- Function Blocks/IOs/Beckhoff/EL2809 - Digital Outputs/DataTypes/EL2809_DEV_CONFIG.TcDUT
TYPE EL2809_DEV_CONFIG :
    STRUCT
       
		enableForce	: BOOL;
		forceDigitalOutput_00 : BOOL;
		forceDigitalOutput_01 : BOOL;
		forceDigitalOutput_02 : BOOL;
		forceDigitalOutput_03 : BOOL;
		forceDigitalOutput_04 : BOOL;
		forceDigitalOutput_05 : BOOL;
		forceDigitalOutput_06 : BOOL;
		forceDigitalOutput_07 : BOOL;
		forceDigitalOutput_08 : BOOL;
		forceDigitalOutput_09 : BOOL;
		forceDigitalOutput_10 : BOOL;
		forceDigitalOutput_11 : BOOL;
		forceDigitalOutput_12 : BOOL;
		forceDigitalOutput_13 : BOOL;
		forceDigitalOutput_14 : BOOL;
		forceDigitalOutput_15 : BOOL;
			


    END_STRUCT
END_TYPE

// ---- Function Blocks/IOs/Beckhoff/EL2809 - Digital Outputs/DataTypes/EL2809_PLCTOHW_PDOS.TcDUT
TYPE EL2809_PLCTOHW_PDOS :
	STRUCT
		
		digitalOutput_01 AT %Q* : BOOL;
		digitalOutput_02 AT %Q* : BOOL;
		digitalOutput_03 AT %Q* : BOOL;
		digitalOutput_04 AT %Q* : BOOL;
		digitalOutput_05 AT %Q* : BOOL;
		digitalOutput_06 AT %Q* : BOOL;
		digitalOutput_07 AT %Q* : BOOL;
		digitalOutput_08 AT %Q* : BOOL;
		digitalOutput_09 AT %Q* : BOOL;
		digitalOutput_10 AT %Q* : BOOL;
		digitalOutput_11 AT %Q* : BOOL;
		digitalOutput_12 AT %Q* : BOOL;
		digitalOutput_13 AT %Q* : BOOL;
		digitalOutput_14 AT %Q* : BOOL;
		digitalOutput_15 AT %Q* : BOOL;
		digitalOutput_16 AT %Q* : BOOL;

	END_STRUCT
END_TYPE

// ---- Function Blocks/IOs/Beckhoff/EL3152 - Ai 2 x 4-20MA - 16bit/DataTypes/EL3152_CHANNEL.TcDUT
TYPE EL3152_CHANNEL :
	STRUCT
		
	
	Status 	AT %I* : EL3152_DEV_STATUS;
	Value 	AT %I* : INT;
	
	
	END_STRUCT
END_TYPE

// ---- Function Blocks/IOs/Beckhoff/EL3152 - Ai 2 x 4-20MA - 16bit/DataTypes/EL3152_DEV_CONFIG.TcDUT
TYPE EL3152_DEV_CONFIG :
    STRUCT
   
        // Setpoint scaling
       	channel1InputLow        : REAL := 0.0;   // Minimum input value for setpoint		
        channel1InputHigh       : REAL := 30518.0; // Maximum input value for setpoint
        channel1OutputLow       : REAL := 0.0; // Minimum output value for setpoint
        channel1OutputHigh      : REAL := 100.0; // Maximum output value for setpoint
        // Setpoint scaling
       	channe12InputLow        : REAL := 0.0;   // Minimum input value for setpoint		
        channe12InputHigh       : REAL := 30518.0; // Maximum input value for setpoint
        channe12OutputLow       : REAL := 0.0; // Minimum output value for setpoint
        channe12OutputHigh      : REAL := 100.0; // Maximum output value for setpoint		

